   instHMISettings.instAniPNTmr.stations.me[24].kp8Config.colorOn1[0] := 'off';
   instHMISettings.instAniPNTmr.stations.me[24].kp8Config.colorOn1[1] := 'off';
   instHMISettings.instAniPNTmr.stations.me[24].kp8Config.colorOn1[2] := 'off';
   instHMISettings.instAniPNTmr.stations.me[24].kp8Config.colorOn1[3] := 'off';
   instHMISettings.instAniPNTmr.stations.me[24].kp8Config.colorOn1[4] := 'off';
   instHMISettings.instAniPNTmr.stations.me[24].kp8Config.colorOn1[5] := 'off';
   instHMISettings.instAniPNTmr.stations.me[24].kp8Config.colorOn1[6] := 'off';
   instHMISettings.instAniPNTmr.stations.me[24].kp8Config.colorOn1[7] := 'yellow';
   instHMISettings.instAniPNTmr.stations.me[24].kp8Config.colorOn2[0] := 'off';
   instHMISettings.instAniPNTmr.stations.me[24].kp8Config.colorOn2[1] := 'off';
   instHMISettings.instAniPNTmr.stations.me[24].kp8Config.colorOn2[2] := 'off';
   instHMISettings.instAniPNTmr.stations.me[24].kp8Config.colorOn2[3] := 'off';
   instHMISettings.instAniPNTmr.stations.me[24].kp8Config.colorOn2[4] := 'off';
   instHMISettings.instAniPNTmr.stations.me[24].kp8Config.colorOn2[5] := 'off';
   instHMISettings.instAniPNTmr.stations.me[24].kp8Config.colorOn2[6] := 'off';
   instHMISettings.instAniPNTmr.stations.me[24].kp8Config.colorOff[0] := 'off';
   instHMISettings.instAniPNTmr.stations.me[24].kp8Config.colorOff[1] := 'off';
   instHMISettings.instAniPNTmr.stations.me[24].kp8Config.colorOff[2] := 'off';
   instHMISettings.instAniPNTmr.stations.me[24].kp8Config.colorOff[3] := 'off';
   instHMISettings.instAniPNTmr.stations.me[24].kp8Config.colorOff[4] := 'off';
   instHMISettings.instAniPNTmr.stations.me[24].kp8Config.colorOff[5] := 'off';
   instHMISettings.instAniPNTmr.stations.me[24].kp8Config.colorOff[6] := 'off';
   instHMISettings.instAniPNTmr.stations.me[24].kp8Config.colorOff[7] := 'green';
   instHMISettings.instAniPNTmr.stations.me[24].kp8Config.mode[7] := TRUE;
   instHMISettings.instAniPNTmr.stations.me[24].kp8Out := 16#0080_0000;
   instHMISettings.instAniPNTmr.stations.me[24].line := WSTRING#'LGS';
   instHMISettings.instAniPNTmr.stations.me[24].partNumbers[0] := WSTRING#'';
   instHMISettings.instAniPNTmr.stations.me[24].partNumbers[1] := WSTRING#'';
   instHMISettings.instAniPNTmr.stations.me[24].partNumbers[2] := WSTRING#'';
   instHMISettings.instAniPNTmr.stations.me[24].partNumbers[3] := WSTRING#'';
   instHMISettings.instAniPNTmr.stations.me[24].partNumbers[4] := WSTRING#'';
   instHMISettings.instAniPNTmr.stations.me[24].partNumbers[5] := WSTRING#'';
   instHMISettings.instAniPNTmr.stations.me[24].partNumbers[6] := WSTRING#'';
   instHMISettings.instAniPNTmr.stations.me[24].partNumbers[7] := WSTRING#'16.08.208.411.030C';
   instHMISettings.instAniPNTmr.stations.me[24].presetTime.allotted[7] := 1800.0;
   instHMISettings.instAniPNTmr.stations.me[24].presetTime.critical[7] := 300.0;
   instHMISettings.instAniPNTmr.stations.me[24].stackLightOut := 16#0400_0000;
   instHMISettings.instAniPNTmr.stations.me[25].btnStates[0] := TRUE;
   instHMISettings.instAniPNTmr.stations.me[25].dropZone := 1;
   instHMISettings.instAniPNTmr.stations.me[25].kp8Config.activate[1] := TRUE;
   instHMISettings.instAniPNTmr.stations.me[25].kp8Config.activate[2] := TRUE;
   instHMISettings.instAniPNTmr.stations.me[25].kp8Config.activate[6] := TRUE;
   instHMISettings.instAniPNTmr.stations.me[25].kp8Config.activate[7] := TRUE;
   instHMISettings.instAniPNTmr.stations.me[25].kp8Config.colorOn1[0] := 'off';
   instHMISettings.instAniPNTmr.stations.me[25].kp8Config.colorOn1[1] := 'yellow';
   instHMISettings.instAniPNTmr.stations.me[25].kp8Config.colorOn1[2] := 'yellow';
   instHMISettings.instAniPNTmr.stations.me[25].kp8Config.colorOn1[3] := 'off';
   instHMISettings.instAniPNTmr.stations.me[25].kp8Config.colorOn1[4] := 'off';
   instHMISettings.instAniPNTmr.stations.me[25].kp8Config.colorOn1[5] := 'off';
   instHMISettings.instAniPNTmr.stations.me[25].kp8Config.colorOn1[6] := 'yellow';
   instHMISettings.instAniPNTmr.stations.me[25].kp8Config.colorOn1[7] := 'yellow';
   instHMISettings.instAniPNTmr.stations.me[25].kp8Config.colorOn2[0] := 'off';
   instHMISettings.instAniPNTmr.stations.me[25].kp8Config.colorOn2[3] := 'off';
   instHMISettings.instAniPNTmr.stations.me[25].kp8Config.colorOn2[4] := 'off';
   instHMISettings.instAniPNTmr.stations.me[25].kp8Config.colorOn2[5] := 'off';
   instHMISettings.instAniPNTmr.stations.me[25].kp8Config.colorOff[0] := 'off';
   instHMISettings.instAniPNTmr.stations.me[25].kp8Config.colorOff[1] := 'green';
   instHMISettings.instAniPNTmr.stations.me[25].kp8Config.colorOff[2] := 'green';
   instHMISettings.instAniPNTmr.stations.me[25].kp8Config.colorOff[3] := 'off';
   instHMISettings.instAniPNTmr.stations.me[25].kp8Config.colorOff[4] := 'off';
   instHMISettings.instAniPNTmr.stations.me[25].kp8Config.colorOff[5] := 'off';
   instHMISettings.instAniPNTmr.stations.me[25].kp8Config.colorOff[6] := 'green';
   instHMISettings.instAniPNTmr.stations.me[25].kp8Config.colorOff[7] := 'green';
   instHMISettings.instAniPNTmr.stations.me[25].kp8Config.mode[1] := TRUE;
   instHMISettings.instAniPNTmr.stations.me[25].kp8Config.mode[2] := TRUE;
   instHMISettings.instAniPNTmr.stations.me[25].kp8Config.mode[6] := TRUE;
   instHMISettings.instAniPNTmr.stations.me[25].kp8Config.mode[7] := TRUE;
   instHMISettings.instAniPNTmr.stations.me[25].kp8Out := 16#4000_8400;
   instHMISettings.instAniPNTmr.stations.me[25].line := WSTRING#'CV';
   instHMISettings.instAniPNTmr.stations.me[25].partNumbers[0] := WSTRING#'';
   instHMISettings.instAniPNTmr.stations.me[25].partNumbers[1] := WSTRING#'C/O MATERIALS';
   instHMISettings.instAniPNTmr.stations.me[25].partNumbers[2] := WSTRING#'16.08.216.806.020A';
   instHMISettings.instAniPNTmr.stations.me[25].partNumbers[3] := WSTRING#'';
   instHMISettings.instAniPNTmr.stations.me[25].partNumbers[4] := WSTRING#'';
   instHMISettings.instAniPNTmr.stations.me[25].partNumbers[5] := WSTRING#'';
   instHMISettings.instAniPNTmr.stations.me[25].partNumbers[6] := WSTRING#'16.08.208.631.000F';
   instHMISettings.instAniPNTmr.stations.me[25].partNumbers[7] := WSTRING#'16.08.216.315.000A';
   instHMISettings.instAniPNTmr.stations.me[25].presetTime.allotted[1] := 1800.0;
   instHMISettings.instAniPNTmr.stations.me[25].presetTime.allotted[2] := 1800.0;
   instHMISettings.instAniPNTmr.stations.me[25].presetTime.allotted[6] := 1800.0;
   instHMISettings.instAniPNTmr.stations.me[25].presetTime.allotted[7] := 1800.0;
   instHMISettings.instAniPNTmr.stations.me[25].presetTime.critical[1] := 300.0;
   instHMISettings.instAniPNTmr.stations.me[25].presetTime.critical[2] := 300.0;
   instHMISettings.instAniPNTmr.stations.me[25].presetTime.critical[6] := 300.0;
   instHMISettings.instAniPNTmr.stations.me[25].presetTime.critical[7] := 300.0;
   instHMISettings.instAniPNTmr.stations.me[25].settings.btnSelection[1] := TRUE;
   instHMISettings.instAniPNTmr.stations.me[25].stackLightOut := 16#0409_0200;
   instHMISettings.instAniPNTmr.stations.me[26].animations[3] := 3;
   instHMISettings.instAniPNTmr.stations.me[26].btnStates[3] := TRUE;
   instHMISettings.instAniPNTmr.stations.me[26].dropZone := 2;
   instHMISettings.instAniPNTmr.stations.me[26].elapsedTime.partReq[3] := 2305.587;
   instHMISettings.instAniPNTmr.stations.me[26].kp8Config.activate[1] := TRUE;
   instHMISettings.instAniPNTmr.stations.me[26].kp8Config.activate[2] := TRUE;
   instHMISettings.instAniPNTmr.stations.me[26].kp8Config.activate[3] := TRUE;
   instHMISettings.instAniPNTmr.stations.me[26].kp8Config.activate[5] := TRUE;
   instHMISettings.instAniPNTmr.stations.me[26].kp8Config.activate[6] := TRUE;
   instHMISettings.instAniPNTmr.stations.me[26].kp8Config.activate[7] := TRUE;
   instHMISettings.instAniPNTmr.stations.me[26].kp8Config.colorOn1[0] := 'off';
   instHMISettings.instAniPNTmr.stations.me[26].kp8Config.colorOn1[1] := 'yellow';
   instHMISettings.instAniPNTmr.stations.me[26].kp8Config.colorOn1[2] := 'yellow';
   instHMISettings.instAniPNTmr.stations.me[26].kp8Config.colorOn1[3] := 'yellow';
   instHMISettings.instAniPNTmr.stations.me[26].kp8Config.colorOn1[4] := 'off';
   instHMISettings.instAniPNTmr.stations.me[26].kp8Config.colorOn1[5] := 'yellow';
   instHMISettings.instAniPNTmr.stations.me[26].kp8Config.colorOn1[6] := 'yellow';
   instHMISettings.instAniPNTmr.stations.me[26].kp8Config.colorOn1[7] := 'yellow';
   instHMISettings.instAniPNTmr.stations.me[26].kp8Config.colorOn2[0] := 'off';
   instHMISettings.instAniPNTmr.stations.me[26].kp8Config.colorOn2[4] := 'off';
   instHMISettings.instAniPNTmr.stations.me[26].kp8Config.colorOff[0] := 'off';
   instHMISettings.instAniPNTmr.stations.me[26].kp8Config.colorOff[1] := 'green';
   instHMISettings.instAniPNTmr.stations.me[26].kp8Config.colorOff[2] := 'green';
   instHMISettings.instAniPNTmr.stations.me[26].kp8Config.colorOff[3] := 'green';
   instHMISettings.instAniPNTmr.stations.me[26].kp8Config.colorOff[4] := 'off';
   instHMISettings.instAniPNTmr.stations.me[26].kp8Config.colorOff[5] := 'green';
   instHMISettings.instAniPNTmr.stations.me[26].kp8Config.colorOff[6] := 'green';
   instHMISettings.instAniPNTmr.stations.me[26].kp8Config.colorOff[7] := 'green';
   instHMISettings.instAniPNTmr.stations.me[26].kp8Config.mode[1] := TRUE;
   instHMISettings.instAniPNTmr.stations.me[26].kp8Config.mode[2] := TRUE;
   instHMISettings.instAniPNTmr.stations.me[26].kp8Config.mode[3] := TRUE;
   instHMISettings.instAniPNTmr.stations.me[26].kp8Config.mode[5] := TRUE;
   instHMISettings.instAniPNTmr.stations.me[26].kp8Config.mode[6] := TRUE;
   instHMISettings.instAniPNTmr.stations.me[26].kp8Config.mode[7] := TRUE;
   instHMISettings.instAniPNTmr.stations.me[26].kp8Out := 16#E000_0000;
   instHMISettings.instAniPNTmr.stations.me[26].line := WSTRING#'CV';
   instHMISettings.instAniPNTmr.stations.me[26].partNumbers[0] := WSTRING#'';
   instHMISettings.instAniPNTmr.stations.me[26].partNumbers[1] := WSTRING#'C/O MATERIALS';
   instHMISettings.instAniPNTmr.stations.me[26].partNumbers[2] := WSTRING#'16.08.216.291.000A';
   instHMISettings.instAniPNTmr.stations.me[26].partNumbers[3] := WSTRING#'16.08.216.315.001A';
   instHMISettings.instAniPNTmr.stations.me[26].partNumbers[4] := WSTRING#'';
   instHMISettings.instAniPNTmr.stations.me[26].partNumbers[5] := WSTRING#'16.08.216.057.001A';
   instHMISettings.instAniPNTmr.stations.me[26].partNumbers[6] := WSTRING#'16.08.208.661.000F';
   instHMISettings.instAniPNTmr.stations.me[26].partNumbers[7] := WSTRING#'16.08.216.315.002A';
   instHMISettings.instAniPNTmr.stations.me[26].partOrdered[3] := TRUE;
   instHMISettings.instAniPNTmr.stations.me[26].partRequested[3] := TRUE;
   instHMISettings.instAniPNTmr.stations.me[26].presetTime.allotted[1] := 1800.0;
   instHMISettings.instAniPNTmr.stations.me[26].presetTime.allotted[2] := 1800.0;
   instHMISettings.instAniPNTmr.stations.me[26].presetTime.allotted[3] := 1800.0;
   instHMISettings.instAniPNTmr.stations.me[26].presetTime.allotted[5] := 1800.0;
   instHMISettings.instAniPNTmr.stations.me[26].presetTime.allotted[6] := 1800.0;
   instHMISettings.instAniPNTmr.stations.me[26].presetTime.allotted[7] := 1800.0;
   instHMISettings.instAniPNTmr.stations.me[26].presetTime.critical[1] := 300.0;
   instHMISettings.instAniPNTmr.stations.me[26].presetTime.critical[2] := 300.0;
   instHMISettings.instAniPNTmr.stations.me[26].presetTime.critical[3] := 300.0;
   instHMISettings.instAniPNTmr.stations.me[26].presetTime.critical[5] := 300.0;
   instHMISettings.instAniPNTmr.stations.me[26].presetTime.critical[6] := 300.0;
   instHMISettings.instAniPNTmr.stations.me[26].presetTime.critical[7] := 300.0;
   instHMISettings.instAniPNTmr.stations.me[26].stackLightOut := 16#0449_0200;
   instHMISettings.instAniPNTmr.stations.me[27].dropZone := 3;
   instHMISettings.instAniPNTmr.stations.me[27].kp8Config.activate[1] := TRUE;
   instHMISettings.instAniPNTmr.stations.me[27].kp8Config.activate[2] := TRUE;
   instHMISettings.instAniPNTmr.stations.me[27].kp8Config.activate[3] := TRUE;
   instHMISettings.instAniPNTmr.stations.me[27].kp8Config.activate[5] := TRUE;
   instHMISettings.instAniPNTmr.stations.me[27].kp8Config.activate[6] := TRUE;
   instHMISettings.instAniPNTmr.stations.me[27].kp8Config.activate[7] := TRUE;
   instHMISettings.instAniPNTmr.stations.me[27].kp8Config.colorOn1[0] := 'off';
   instHMISettings.instAniPNTmr.stations.me[27].kp8Config.colorOn1[1] := 'yellow';
   instHMISettings.instAniPNTmr.stations.me[27].kp8Config.colorOn1[2] := 'yellow';
   instHMISettings.instAniPNTmr.stations.me[27].kp8Config.colorOn1[3] := 'yellow';
   instHMISettings.instAniPNTmr.stations.me[27].kp8Config.colorOn1[4] := 'off';
   instHMISettings.instAniPNTmr.stations.me[27].kp8Config.colorOn1[5] := 'yellow';
   instHMISettings.instAniPNTmr.stations.me[27].kp8Config.colorOn1[6] := 'yellow';
   instHMISettings.instAniPNTmr.stations.me[27].kp8Config.colorOn1[7] := 'yellow';
   instHMISettings.instAniPNTmr.stations.me[27].kp8Config.colorOn2[0] := 'off';
   instHMISettings.instAniPNTmr.stations.me[27].kp8Config.colorOn2[4] := 'off';
   instHMISettings.instAniPNTmr.stations.me[27].kp8Config.colorOff[0] := 'off';
   instHMISettings.instAniPNTmr.stations.me[27].kp8Config.colorOff[1] := 'green';
   instHMISettings.instAniPNTmr.stations.me[27].kp8Config.colorOff[2] := 'green';
   instHMISettings.instAniPNTmr.stations.me[27].kp8Config.colorOff[3] := 'green';
   instHMISettings.instAniPNTmr.stations.me[27].kp8Config.colorOff[4] := 'off';
   instHMISettings.instAniPNTmr.stations.me[27].kp8Config.colorOff[5] := 'green';
   instHMISettings.instAniPNTmr.stations.me[27].kp8Config.colorOff[6] := 'green';
   instHMISettings.instAniPNTmr.stations.me[27].kp8Config.colorOff[7] := 'green';
   instHMISettings.instAniPNTmr.stations.me[27].kp8Config.mode[1] := TRUE;
   instHMISettings.instAniPNTmr.stations.me[27].kp8Config.mode[2] := TRUE;
   instHMISettings.instAniPNTmr.stations.me[27].kp8Config.mode[3] := TRUE;
   instHMISettings.instAniPNTmr.stations.me[27].kp8Config.mode[5] := TRUE;
   instHMISettings.instAniPNTmr.stations.me[27].kp8Config.mode[6] := TRUE;
   instHMISettings.instAniPNTmr.stations.me[27].kp8Config.mode[7] := TRUE;
   instHMISettings.instAniPNTmr.stations.me[27].kp8Out := 16#4000_A800;
   instHMISettings.instAniPNTmr.stations.me[27].line := WSTRING#'CV';
   instHMISettings.instAniPNTmr.stations.me[27].partNumbers[0] := WSTRING#'';
   instHMISettings.instAniPNTmr.stations.me[27].partNumbers[1] := WSTRING#'C/O MATERIALS';
   instHMISettings.instAniPNTmr.stations.me[27].partNumbers[2] := WSTRING#'16.18.011.301.010A';
   instHMISettings.instAniPNTmr.stations.me[27].partNumbers[3] := WSTRING#'16.18.011.301.020B';
   instHMISettings.instAniPNTmr.stations.me[27].partNumbers[4] := WSTRING#'';
   instHMISettings.instAniPNTmr.stations.me[27].partNumbers[5] := WSTRING#'16.18.007.311.010A';
   instHMISettings.instAniPNTmr.stations.me[27].partNumbers[6] := WSTRING#'16.18.007.311.020A';
   instHMISettings.instAniPNTmr.stations.me[27].partNumbers[7] := WSTRING#'16.18.012.401.020A';
   instHMISettings.instAniPNTmr.stations.me[27].presetTime.allotted[1] := 1800.0;
   instHMISettings.instAniPNTmr.stations.me[27].presetTime.allotted[2] := 1800.0;
   instHMISettings.instAniPNTmr.stations.me[27].presetTime.allotted[3] := 1800.0;
   instHMISettings.instAniPNTmr.stations.me[27].presetTime.allotted[5] := 1800.0;
   instHMISettings.instAniPNTmr.stations.me[27].presetTime.allotted[6] := 1800.0;
   instHMISettings.instAniPNTmr.stations.me[27].presetTime.allotted[7] := 1800.0;
   instHMISettings.instAniPNTmr.stations.me[27].presetTime.critical[1] := 300.0;
   instHMISettings.instAniPNTmr.stations.me[27].presetTime.critical[2] := 300.0;
   instHMISettings.instAniPNTmr.stations.me[27].presetTime.critical[3] := 300.0;
   instHMISettings.instAniPNTmr.stations.me[27].presetTime.critical[5] := 300.0;
   instHMISettings.instAniPNTmr.stations.me[27].presetTime.critical[6] := 300.0;
   instHMISettings.instAniPNTmr.stations.me[27].presetTime.critical[7] := 300.0;
   instHMISettings.instAniPNTmr.stations.me[27].stackLightOut := 16#2449_0200;
   instHMISettings.instAniPNTmr.stations.me[28].dropZone := 4;
   instHMISettings.instAniPNTmr.stations.me[28].kp8Config.activate[1] := TRUE;
   instHMISettings.instAniPNTmr.stations.me[28].kp8Config.activate[3] := TRUE;
   instHMISettings.instAniPNTmr.stations.me[28].kp8Config.activate[6] := TRUE;
   instHMISettings.instAniPNTmr.stations.me[28].kp8Config.activate[7] := TRUE;
   instHMISettings.instAniPNTmr.stations.me[28].kp8Config.colorOn1[0] := 'off';
   instHMISettings.instAniPNTmr.stations.me[28].kp8Config.colorOn1[1] := 'yellow';
   instHMISettings.instAniPNTmr.stations.me[28].kp8Config.colorOn1[2] := 'off';
   instHMISettings.instAniPNTmr.stations.me[28].kp8Config.colorOn1[3] := 'yellow';
   instHMISettings.instAniPNTmr.stations.me[28].kp8Config.colorOn1[4] := 'off';
   instHMISettings.instAniPNTmr.stations.me[28].kp8Config.colorOn1[5] := 'off';
   instHMISettings.instAniPNTmr.stations.me[28].kp8Config.colorOn1[6] := 'yellow';
   instHMISettings.instAniPNTmr.stations.me[28].kp8Config.colorOn1[7] := 'yellow';
   instHMISettings.instAniPNTmr.stations.me[28].kp8Config.colorOn2[0] := 'off';
   instHMISettings.instAniPNTmr.stations.me[28].kp8Config.colorOn2[2] := 'off';
   instHMISettings.instAniPNTmr.stations.me[28].kp8Config.colorOn2[4] := 'off';
   instHMISettings.instAniPNTmr.stations.me[28].kp8Config.colorOn2[5] := 'off';
   instHMISettings.instAniPNTmr.stations.me[28].kp8Config.colorOff[0] := 'off';
   instHMISettings.instAniPNTmr.stations.me[28].kp8Config.colorOff[1] := 'green';
   instHMISettings.instAniPNTmr.stations.me[28].kp8Config.colorOff[2] := 'off';
   instHMISettings.instAniPNTmr.stations.me[28].kp8Config.colorOff[3] := 'green';
   instHMISettings.instAniPNTmr.stations.me[28].kp8Config.colorOff[4] := 'off';
   instHMISettings.instAniPNTmr.stations.me[28].kp8Config.colorOff[5] := 'off';
   instHMISettings.instAniPNTmr.stations.me[28].kp8Config.colorOff[6] := 'green';
   instHMISettings.instAniPNTmr.stations.me[28].kp8Config.colorOff[7] := 'green';
   instHMISettings.instAniPNTmr.stations.me[28].kp8Config.mode[1] := TRUE;
   instHMISettings.instAniPNTmr.stations.me[28].kp8Config.mode[3] := TRUE;
   instHMISettings.instAniPNTmr.stations.me[28].kp8Config.mode[6] := TRUE;
   instHMISettings.instAniPNTmr.stations.me[28].kp8Config.mode[7] := TRUE;
   instHMISettings.instAniPNTmr.stations.me[28].kp8Out := 16#0000_6E00;
   instHMISettings.instAniPNTmr.stations.me[28].line := WSTRING#'CV';
   instHMISettings.instAniPNTmr.stations.me[28].partNumbers[0] := WSTRING#'';
   instHMISettings.instAniPNTmr.stations.me[28].partNumbers[1] := WSTRING#'C/O MATERIALS';
   instHMISettings.instAniPNTmr.stations.me[28].partNumbers[2] := WSTRING#'';
   instHMISettings.instAniPNTmr.stations.me[28].partNumbers[3] := WSTRING#'16.32.112.543.210E';
   instHMISettings.instAniPNTmr.stations.me[28].partNumbers[4] := WSTRING#'';
   instHMISettings.instAniPNTmr.stations.me[28].partNumbers[5] := WSTRING#'';
   instHMISettings.instAniPNTmr.stations.me[28].partNumbers[6] := WSTRING#'16.32.112.543.020A';
   instHMISettings.instAniPNTmr.stations.me[28].partNumbers[7] := WSTRING#'16.32.112.315.018A';
   instHMISettings.instAniPNTmr.stations.me[28].presetTime.allotted[1] := 1800.0;
   instHMISettings.instAniPNTmr.stations.me[28].presetTime.allotted[3] := 1800.0;
   instHMISettings.instAniPNTmr.stations.me[28].presetTime.allotted[6] := 1800.0;
   instHMISettings.instAniPNTmr.stations.me[28].presetTime.allotted[7] := 1800.0;
   instHMISettings.instAniPNTmr.stations.me[28].presetTime.critical[1] := 300.0;
   instHMISettings.instAniPNTmr.stations.me[28].presetTime.critical[3] := 300.0;
   instHMISettings.instAniPNTmr.stations.me[28].presetTime.critical[6] := 300.0;
   instHMISettings.instAniPNTmr.stations.me[28].presetTime.critical[7] := 300.0;
   instHMISettings.instAniPNTmr.stations.me[28].stackLightOut := 16#2401_0200;
   instHMISettings.instAniPNTmr.stations.me[29].dropZone := 1;
   instHMISettings.instAniPNTmr.stations.me[29].kp8Config.activate[1] := TRUE;
   instHMISettings.instAniPNTmr.stations.me[29].kp8Config.activate[2] := TRUE;
   instHMISettings.instAniPNTmr.stations.me[29].kp8Config.activate[3] := TRUE;
   instHMISettings.instAniPNTmr.stations.me[29].kp8Config.activate[5] := TRUE;
   instHMISettings.instAniPNTmr.stations.me[29].kp8Config.activate[6] := TRUE;
   instHMISettings.instAniPNTmr.stations.me[29].kp8Config.activate[7] := TRUE;
   instHMISettings.instAniPNTmr.stations.me[29].kp8Config.colorOn1[0] := 'off';
   instHMISettings.instAniPNTmr.stations.me[29].kp8Config.colorOn1[1] := 'yellow';
   instHMISettings.instAniPNTmr.stations.me[29].kp8Config.colorOn1[2] := 'yellow';
   instHMISettings.instAniPNTmr.stations.me[29].kp8Config.colorOn1[3] := 'yellow';
   instHMISettings.instAniPNTmr.stations.me[29].kp8Config.colorOn1[4] := 'off';
   instHMISettings.instAniPNTmr.stations.me[29].kp8Config.colorOn1[5] := 'yellow';
   instHMISettings.instAniPNTmr.stations.me[29].kp8Config.colorOn1[6] := 'yellow';
   instHMISettings.instAniPNTmr.stations.me[29].kp8Config.colorOn1[7] := 'yellow';
   instHMISettings.instAniPNTmr.stations.me[29].kp8Config.colorOn2[0] := 'off';
   instHMISettings.instAniPNTmr.stations.me[29].kp8Config.colorOn2[4] := 'off';
   instHMISettings.instAniPNTmr.stations.me[29].kp8Config.colorOff[0] := 'off';
   instHMISettings.instAniPNTmr.stations.me[29].kp8Config.colorOff[1] := 'green';
   instHMISettings.instAniPNTmr.stations.me[29].kp8Config.colorOff[2] := 'green';
   instHMISettings.instAniPNTmr.stations.me[29].kp8Config.colorOff[3] := 'green';
   instHMISettings.instAniPNTmr.stations.me[29].kp8Config.colorOff[4] := 'off';
   instHMISettings.instAniPNTmr.stations.me[29].kp8Config.colorOff[5] := 'green';
   instHMISettings.instAniPNTmr.stations.me[29].kp8Config.colorOff[6] := 'green';
   instHMISettings.instAniPNTmr.stations.me[29].kp8Config.colorOff[7] := 'green';
   instHMISettings.instAniPNTmr.stations.me[29].kp8Config.mode[1] := TRUE;
   instHMISettings.instAniPNTmr.stations.me[29].kp8Config.mode[2] := TRUE;
   instHMISettings.instAniPNTmr.stations.me[29].kp8Config.mode[3] := TRUE;
   instHMISettings.instAniPNTmr.stations.me[29].kp8Config.mode[5] := TRUE;
   instHMISettings.instAniPNTmr.stations.me[29].kp8Config.mode[6] := TRUE;
   instHMISettings.instAniPNTmr.stations.me[29].kp8Config.mode[7] := TRUE;
   instHMISettings.instAniPNTmr.stations.me[29].kp8Out := 16#2A00_4400;
   instHMISettings.instAniPNTmr.stations.me[29].line := WSTRING#'PC';
   instHMISettings.instAniPNTmr.stations.me[29].partNumbers[0] := WSTRING#'';
   instHMISettings.instAniPNTmr.stations.me[29].partNumbers[1] := WSTRING#'C/O MATERIALS';
   instHMISettings.instAniPNTmr.stations.me[29].partNumbers[2] := WSTRING#'11.54.007.052.007B';
   instHMISettings.instAniPNTmr.stations.me[29].partNumbers[3] := WSTRING#'11.54.007.315.026G';
   instHMISettings.instAniPNTmr.stations.me[29].partNumbers[4] := WSTRING#'';
   instHMISettings.instAniPNTmr.stations.me[29].partNumbers[5] := WSTRING#'11.54.007.052.008A';
   instHMISettings.instAniPNTmr.stations.me[29].partNumbers[6] := WSTRING#'11.54.007.045.015D';
   instHMISettings.instAniPNTmr.stations.me[29].partNumbers[7] := WSTRING#'11.54.017.315.001F';
   instHMISettings.instAniPNTmr.stations.me[29].presetTime.allotted[1] := 1800.0;
   instHMISettings.instAniPNTmr.stations.me[29].presetTime.allotted[2] := 1800.0;
   instHMISettings.instAniPNTmr.stations.me[29].presetTime.allotted[3] := 1800.0;
   instHMISettings.instAniPNTmr.stations.me[29].presetTime.allotted[5] := 1800.0;
   instHMISettings.instAniPNTmr.stations.me[29].presetTime.allotted[6] := 1800.0;
   instHMISettings.instAniPNTmr.stations.me[29].presetTime.allotted[7] := 1800.0;
   instHMISettings.instAniPNTmr.stations.me[29].presetTime.critical[1] := 300.0;
   instHMISettings.instAniPNTmr.stations.me[29].presetTime.critical[2] := 300.0;
   instHMISettings.instAniPNTmr.stations.me[29].presetTime.critical[3] := 300.0;
   instHMISettings.instAniPNTmr.stations.me[29].presetTime.critical[5] := 300.0;
   instHMISettings.instAniPNTmr.stations.me[29].presetTime.critical[6] := 300.0;
   instHMISettings.instAniPNTmr.stations.me[29].presetTime.critical[7] := 300.0;
   instHMISettings.instAniPNTmr.stations.me[29].settings.btnSelection[3] := TRUE;
   instHMISettings.instAniPNTmr.stations.me[29].stackLightOut := 16#2449_0200;
   instHMISettings.instAniPNTmr.stations.me[30].dropZone := 1;
   instHMISettings.instAniPNTmr.stations.me[30].kp8Config.activate[7] := TRUE;
   instHMISettings.instAniPNTmr.stations.me[30].kp8Config.colorOn1[0] := 'off';
   instHMISettings.instAniPNTmr.stations.me[30].kp8Config.colorOn1[1] := 'off';
   instHMISettings.instAniPNTmr.stations.me[30].kp8Config.colorOn1[2] := 'off';
   instHMISettings.instAniPNTmr.stations.me[30].kp8Config.colorOn1[3] := 'off';
   instHMISettings.instAniPNTmr.stations.me[30].kp8Config.colorOn1[4] := 'off';
   instHMISettings.instAniPNTmr.stations.me[30].kp8Config.colorOn1[5] := 'off';
   instHMISettings.instAniPNTmr.stations.me[30].kp8Config.colorOn1[6] := 'off';
   instHMISettings.instAniPNTmr.stations.me[30].kp8Config.colorOn1[7] := 'yellow';
   instHMISettings.instAniPNTmr.stations.me[30].kp8Config.colorOn2[0] := 'off';
   instHMISettings.instAniPNTmr.stations.me[30].kp8Config.colorOn2[1] := 'off';
   instHMISettings.instAniPNTmr.stations.me[30].kp8Config.colorOn2[2] := 'off';
   instHMISettings.instAniPNTmr.stations.me[30].kp8Config.colorOn2[3] := 'off';
   instHMISettings.instAniPNTmr.stations.me[30].kp8Config.colorOn2[4] := 'off';
   instHMISettings.instAniPNTmr.stations.me[30].kp8Config.colorOn2[5] := 'off';
   instHMISettings.instAniPNTmr.stations.me[30].kp8Config.colorOn2[6] := 'off';
   instHMISettings.instAniPNTmr.stations.me[30].kp8Config.colorOff[0] := 'off';
   instHMISettings.instAniPNTmr.stations.me[30].kp8Config.colorOff[1] := 'off';
   instHMISettings.instAniPNTmr.stations.me[30].kp8Config.colorOff[2] := 'off';
   instHMISettings.instAniPNTmr.stations.me[30].kp8Config.colorOff[3] := 'off';
   instHMISettings.instAniPNTmr.stations.me[30].kp8Config.colorOff[4] := 'off';
   instHMISettings.instAniPNTmr.stations.me[30].kp8Config.colorOff[5] := 'off';
   instHMISettings.instAniPNTmr.stations.me[30].kp8Config.colorOff[6] := 'off';
   instHMISettings.instAniPNTmr.stations.me[30].kp8Config.colorOff[7] := 'green';
   instHMISettings.instAniPNTmr.stations.me[30].kp8Config.mode[7] := TRUE;
   instHMISettings.instAniPNTmr.stations.me[30].kp8Out := 16#0080_0000;
   instHMISettings.instAniPNTmr.stations.me[30].line := WSTRING#'VN127';
   instHMISettings.instAniPNTmr.stations.me[30].partNumbers[0] := WSTRING#'';
   instHMISettings.instAniPNTmr.stations.me[30].partNumbers[1] := WSTRING#'';
   instHMISettings.instAniPNTmr.stations.me[30].partNumbers[2] := WSTRING#'';
   instHMISettings.instAniPNTmr.stations.me[30].partNumbers[3] := WSTRING#'';
   instHMISettings.instAniPNTmr.stations.me[30].partNumbers[4] := WSTRING#'';
   instHMISettings.instAniPNTmr.stations.me[30].partNumbers[5] := WSTRING#'';
   instHMISettings.instAniPNTmr.stations.me[30].partNumbers[6] := WSTRING#'';
   instHMISettings.instAniPNTmr.stations.me[30].partNumbers[7] := WSTRING#'11.54.313.872.000E';
   instHMISettings.instAniPNTmr.stations.me[30].presetTime.allotted[7] := 1800.0;
   instHMISettings.instAniPNTmr.stations.me[30].presetTime.critical[7] := 300.0;
   instHMISettings.instAniPNTmr.stations.me[30].settings.btnSelection[7] := TRUE;
   instHMISettings.instAniPNTmr.stations.me[30].stackLightOut := 16#0400_0000;
   instHMISettings.instAniPNTmr.stations.me[31].dropZone := 1;
   instHMISettings.instAniPNTmr.stations.me[31].kp8Config.activate[3] := TRUE;
   instHMISettings.instAniPNTmr.stations.me[31].kp8Config.activate[7] := TRUE;
   instHMISettings.instAniPNTmr.stations.me[31].kp8Config.colorOn1[0] := 'off';
   instHMISettings.instAniPNTmr.stations.me[31].kp8Config.colorOn1[1] := 'off';
   instHMISettings.instAniPNTmr.stations.me[31].kp8Config.colorOn1[2] := 'off';
   instHMISettings.instAniPNTmr.stations.me[31].kp8Config.colorOn1[3] := 'yellow';
   instHMISettings.instAniPNTmr.stations.me[31].kp8Config.colorOn1[4] := 'off';
   instHMISettings.instAniPNTmr.stations.me[31].kp8Config.colorOn1[5] := 'off';
   instHMISettings.instAniPNTmr.stations.me[31].kp8Config.colorOn1[6] := 'off';
   instHMISettings.instAniPNTmr.stations.me[31].kp8Config.colorOn1[7] := 'yellow';
   instHMISettings.instAniPNTmr.stations.me[31].kp8Config.colorOn2[0] := 'off';
   instHMISettings.instAniPNTmr.stations.me[31].kp8Config.colorOn2[1] := 'off';
   instHMISettings.instAniPNTmr.stations.me[31].kp8Config.colorOn2[2] := 'off';
   instHMISettings.instAniPNTmr.stations.me[31].kp8Config.colorOn2[4] := 'off';
   instHMISettings.instAniPNTmr.stations.me[31].kp8Config.colorOn2[5] := 'off';
   instHMISettings.instAniPNTmr.stations.me[31].kp8Config.colorOn2[6] := 'off';
   instHMISettings.instAniPNTmr.stations.me[31].kp8Config.colorOff[0] := 'off';
   instHMISettings.instAniPNTmr.stations.me[31].kp8Config.colorOff[1] := 'off';
   instHMISettings.instAniPNTmr.stations.me[31].kp8Config.colorOff[2] := 'off';
   instHMISettings.instAniPNTmr.stations.me[31].kp8Config.colorOff[3] := 'green';
   instHMISettings.instAniPNTmr.stations.me[31].kp8Config.colorOff[4] := 'off';
   instHMISettings.instAniPNTmr.stations.me[31].kp8Config.colorOff[5] := 'off';
   instHMISettings.instAniPNTmr.stations.me[31].kp8Config.colorOff[6] := 'off';
   instHMISettings.instAniPNTmr.stations.me[31].kp8Config.colorOff[7] := 'green';
   instHMISettings.instAniPNTmr.stations.me[31].kp8Config.mode[3] := TRUE;
   instHMISettings.instAniPNTmr.stations.me[31].kp8Config.mode[7] := TRUE;
   instHMISettings.instAniPNTmr.stations.me[31].kp8Out := 16#0088_0000;
   instHMISettings.instAniPNTmr.stations.me[31].line := WSTRING#'1BX 2.0';
   instHMISettings.instAniPNTmr.stations.me[31].partNumbers[0] := WSTRING#'';
   instHMISettings.instAniPNTmr.stations.me[31].partNumbers[1] := WSTRING#'';
   instHMISettings.instAniPNTmr.stations.me[31].partNumbers[2] := WSTRING#'';
   instHMISettings.instAniPNTmr.stations.me[31].partNumbers[3] := WSTRING#'16.08.216.011.030B';
   instHMISettings.instAniPNTmr.stations.me[31].partNumbers[4] := WSTRING#'';
   instHMISettings.instAniPNTmr.stations.me[31].partNumbers[5] := WSTRING#'';
   instHMISettings.instAniPNTmr.stations.me[31].partNumbers[6] := WSTRING#'';
   instHMISettings.instAniPNTmr.stations.me[31].partNumbers[7] := WSTRING#'16.08.208.161.030E';
   instHMISettings.instAniPNTmr.stations.me[31].presetTime.allotted[3] := 1800.0;
   instHMISettings.instAniPNTmr.stations.me[31].presetTime.allotted[7] := 1800.0;
   instHMISettings.instAniPNTmr.stations.me[31].presetTime.critical[3] := 300.0;
   instHMISettings.instAniPNTmr.stations.me[31].presetTime.critical[7] := 300.0;
   instHMISettings.instAniPNTmr.stations.me[31].stackLightOut := 16#2400_0000;
   instHMISettings.instAniPNTmr.stations.me[32].dropZone := 2;
   instHMISettings.instAniPNTmr.stations.me[32].kp8Config.activate[7] := TRUE;
   instHMISettings.instAniPNTmr.stations.me[32].kp8Config.colorOn1[0] := 'off';
   instHMISettings.instAniPNTmr.stations.me[32].kp8Config.colorOn1[1] := 'off';
   instHMISettings.instAniPNTmr.stations.me[32].kp8Config.colorOn1[2] := 'off';
   instHMISettings.instAniPNTmr.stations.me[32].kp8Config.colorOn1[3] := 'off';
   instHMISettings.instAniPNTmr.stations.me[32].kp8Config.colorOn1[4] := 'off';
   instHMISettings.instAniPNTmr.stations.me[32].kp8Config.colorOn1[5] := 'off';
   instHMISettings.instAniPNTmr.stations.me[32].kp8Config.colorOn1[6] := 'off';
   instHMISettings.instAniPNTmr.stations.me[32].kp8Config.colorOn1[7] := 'yellow';
   instHMISettings.instAniPNTmr.stations.me[32].kp8Config.colorOn2[0] := 'off';
   instHMISettings.instAniPNTmr.stations.me[32].kp8Config.colorOn2[1] := 'off';
   instHMISettings.instAniPNTmr.stations.me[32].kp8Config.colorOn2[2] := 'off';
   instHMISettings.instAniPNTmr.stations.me[32].kp8Config.colorOn2[3] := 'off';
   instHMISettings.instAniPNTmr.stations.me[32].kp8Config.colorOn2[4] := 'off';
   instHMISettings.instAniPNTmr.stations.me[32].kp8Config.colorOn2[5] := 'off';
   instHMISettings.instAniPNTmr.stations.me[32].kp8Config.colorOn2[6] := 'off';
   instHMISettings.instAniPNTmr.stations.me[32].kp8Config.colorOff[0] := 'off';
   instHMISettings.instAniPNTmr.stations.me[32].kp8Config.colorOff[1] := 'off';
   instHMISettings.instAniPNTmr.stations.me[32].kp8Config.colorOff[2] := 'off';
   instHMISettings.instAniPNTmr.stations.me[32].kp8Config.colorOff[3] := 'off';
   instHMISettings.instAniPNTmr.stations.me[32].kp8Config.colorOff[4] := 'off';
   instHMISettings.instAniPNTmr.stations.me[32].kp8Config.colorOff[5] := 'off';
   instHMISettings.instAniPNTmr.stations.me[32].kp8Config.colorOff[6] := 'off';
   instHMISettings.instAniPNTmr.stations.me[32].kp8Config.colorOff[7] := 'green';
   instHMISettings.instAniPNTmr.stations.me[32].kp8Config.mode[7] := TRUE;
   instHMISettings.instAniPNTmr.stations.me[32].kp8Out := 16#0080_0000;
   instHMISettings.instAniPNTmr.stations.me[32].line := WSTRING#'1BX 2.0';
   instHMISettings.instAniPNTmr.stations.me[32].partNumbers[0] := WSTRING#'';
   instHMISettings.instAniPNTmr.stations.me[32].partNumbers[1] := WSTRING#'';
   instHMISettings.instAniPNTmr.stations.me[32].partNumbers[2] := WSTRING#'';
   instHMISettings.instAniPNTmr.stations.me[32].partNumbers[3] := WSTRING#'';
   instHMISettings.instAniPNTmr.stations.me[32].partNumbers[4] := WSTRING#'';
   instHMISettings.instAniPNTmr.stations.me[32].partNumbers[5] := WSTRING#'';
   instHMISettings.instAniPNTmr.stations.me[32].partNumbers[6] := WSTRING#'';
   instHMISettings.instAniPNTmr.stations.me[32].partNumbers[7] := WSTRING#'16.08.208.601.010D';
   instHMISettings.instAniPNTmr.stations.me[32].presetTime.allotted[7] := 1800.0;
   instHMISettings.instAniPNTmr.stations.me[32].presetTime.critical[7] := 300.0;
   instHMISettings.instAniPNTmr.stations.me[32].stackLightOut := 16#0400_0000;
   instHMISettings.instAniPNTmr.stations.me[33].dropZone := 3;
   instHMISettings.instAniPNTmr.stations.me[33].kp8Config.activate[7] := TRUE;
   instHMISettings.instAniPNTmr.stations.me[33].kp8Config.colorOn1[0] := 'off';
   instHMISettings.instAniPNTmr.stations.me[33].kp8Config.colorOn1[1] := 'off';
   instHMISettings.instAniPNTmr.stations.me[33].kp8Config.colorOn1[2] := 'off';
   instHMISettings.instAniPNTmr.stations.me[33].kp8Config.colorOn1[3] := 'off';
   instHMISettings.instAniPNTmr.stations.me[33].kp8Config.colorOn1[4] := 'off';
   instHMISettings.instAniPNTmr.stations.me[33].kp8Config.colorOn1[5] := 'off';
   instHMISettings.instAniPNTmr.stations.me[33].kp8Config.colorOn1[6] := 'off';
   instHMISettings.instAniPNTmr.stations.me[33].kp8Config.colorOn1[7] := 'yellow';
   instHMISettings.instAniPNTmr.stations.me[33].kp8Config.colorOn2[0] := 'off';
   instHMISettings.instAniPNTmr.stations.me[33].kp8Config.colorOn2[1] := 'off';
   instHMISettings.instAniPNTmr.stations.me[33].kp8Config.colorOn2[2] := 'off';
   instHMISettings.instAniPNTmr.stations.me[33].kp8Config.colorOn2[3] := 'off';
   instHMISettings.instAniPNTmr.stations.me[33].kp8Config.colorOn2[4] := 'off';
   instHMISettings.instAniPNTmr.stations.me[33].kp8Config.colorOn2[5] := 'off';
   instHMISettings.instAniPNTmr.stations.me[33].kp8Config.colorOn2[6] := 'off';
   instHMISettings.instAniPNTmr.stations.me[33].kp8Config.colorOff[0] := 'off';
   instHMISettings.instAniPNTmr.stations.me[33].kp8Config.colorOff[1] := 'off';
   instHMISettings.instAniPNTmr.stations.me[33].kp8Config.colorOff[2] := 'off';
   instHMISettings.instAniPNTmr.stations.me[33].kp8Config.colorOff[3] := 'off';
   instHMISettings.instAniPNTmr.stations.me[33].kp8Config.colorOff[4] := 'off';
   instHMISettings.instAniPNTmr.stations.me[33].kp8Config.colorOff[5] := 'off';
   instHMISettings.instAniPNTmr.stations.me[33].kp8Config.colorOff[6] := 'off';
   instHMISettings.instAniPNTmr.stations.me[33].kp8Config.colorOff[7] := 'green';
   instHMISettings.instAniPNTmr.stations.me[33].kp8Config.mode[7] := TRUE;
   instHMISettings.instAniPNTmr.stations.me[33].kp8Out := 16#0080_0000;
   instHMISettings.instAniPNTmr.stations.me[33].line := WSTRING#'1BX 2.0';
   instHMISettings.instAniPNTmr.stations.me[33].partNumbers[0] := WSTRING#'';
   instHMISettings.instAniPNTmr.stations.me[33].partNumbers[1] := WSTRING#'';
   instHMISettings.instAniPNTmr.stations.me[33].partNumbers[2] := WSTRING#'';
   instHMISettings.instAniPNTmr.stations.me[33].partNumbers[3] := WSTRING#'';
   instHMISettings.instAniPNTmr.stations.me[33].partNumbers[4] := WSTRING#'';
   instHMISettings.instAniPNTmr.stations.me[33].partNumbers[5] := WSTRING#'';
   instHMISettings.instAniPNTmr.stations.me[33].partNumbers[6] := WSTRING#'';
   instHMISettings.instAniPNTmr.stations.me[33].partNumbers[7] := WSTRING#'16.08.208.691.010D';
   instHMISettings.instAniPNTmr.stations.me[33].presetTime.allotted[7] := 1800.0;
   instHMISettings.instAniPNTmr.stations.me[33].presetTime.critical[7] := 300.0;
   instHMISettings.instAniPNTmr.stations.me[33].stackLightOut := 16#0400_0000;
   instHMISettings.instAniPNTmr.stations.me[34].dropZone := 4;
   instHMISettings.instAniPNTmr.stations.me[34].kp8Config.activate[3] := TRUE;
   instHMISettings.instAniPNTmr.stations.me[34].kp8Config.activate[7] := TRUE;
   instHMISettings.instAniPNTmr.stations.me[34].kp8Config.colorOn1[0] := 'off';
   instHMISettings.instAniPNTmr.stations.me[34].kp8Config.colorOn1[1] := 'off';
   instHMISettings.instAniPNTmr.stations.me[34].kp8Config.colorOn1[2] := 'off';
   instHMISettings.instAniPNTmr.stations.me[34].kp8Config.colorOn1[3] := 'yellow';
   instHMISettings.instAniPNTmr.stations.me[34].kp8Config.colorOn1[4] := 'off';
   instHMISettings.instAniPNTmr.stations.me[34].kp8Config.colorOn1[5] := 'off';
   instHMISettings.instAniPNTmr.stations.me[34].kp8Config.colorOn1[6] := 'off';
   instHMISettings.instAniPNTmr.stations.me[34].kp8Config.colorOn1[7] := 'yellow';
   instHMISettings.instAniPNTmr.stations.me[34].kp8Config.colorOn2[0] := 'off';
   instHMISettings.instAniPNTmr.stations.me[34].kp8Config.colorOn2[1] := 'off';
   instHMISettings.instAniPNTmr.stations.me[34].kp8Config.colorOn2[2] := 'off';
   instHMISettings.instAniPNTmr.stations.me[34].kp8Config.colorOn2[4] := 'off';
   instHMISettings.instAniPNTmr.stations.me[34].kp8Config.colorOn2[5] := 'off';
   instHMISettings.instAniPNTmr.stations.me[34].kp8Config.colorOn2[6] := 'off';
   instHMISettings.instAniPNTmr.stations.me[34].kp8Config.colorOff[0] := 'off';
   instHMISettings.instAniPNTmr.stations.me[34].kp8Config.colorOff[1] := 'off';
   instHMISettings.instAniPNTmr.stations.me[34].kp8Config.colorOff[2] := 'off';
   instHMISettings.instAniPNTmr.stations.me[34].kp8Config.colorOff[3] := 'green';
   instHMISettings.instAniPNTmr.stations.me[34].kp8Config.colorOff[4] := 'off';
   instHMISettings.instAniPNTmr.stations.me[34].kp8Config.colorOff[5] := 'off';
   instHMISettings.instAniPNTmr.stations.me[34].kp8Config.colorOff[6] := 'off';
   instHMISettings.instAniPNTmr.stations.me[34].kp8Config.colorOff[7] := 'green';
   instHMISettings.instAniPNTmr.stations.me[34].kp8Config.mode[3] := TRUE;
   instHMISettings.instAniPNTmr.stations.me[34].kp8Config.mode[7] := TRUE;
   instHMISettings.instAniPNTmr.stations.me[34].kp8Out := 16#0088_0000;
   instHMISettings.instAniPNTmr.stations.me[34].line := WSTRING#'1BX 2.0';
   instHMISettings.instAniPNTmr.stations.me[34].partNumbers[0] := WSTRING#'';
   instHMISettings.instAniPNTmr.stations.me[34].partNumbers[1] := WSTRING#'';
   instHMISettings.instAniPNTmr.stations.me[34].partNumbers[2] := WSTRING#'';
   instHMISettings.instAniPNTmr.stations.me[34].partNumbers[3] := WSTRING#'16.08.208.161.030E';
   instHMISettings.instAniPNTmr.stations.me[34].partNumbers[4] := WSTRING#'';
   instHMISettings.instAniPNTmr.stations.me[34].partNumbers[5] := WSTRING#'';
   instHMISettings.instAniPNTmr.stations.me[34].partNumbers[6] := WSTRING#'';
   instHMISettings.instAniPNTmr.stations.me[34].partNumbers[7] := WSTRING#'16.08.216.011.030B';
   instHMISettings.instAniPNTmr.stations.me[34].presetTime.allotted[3] := 1800.0;
   instHMISettings.instAniPNTmr.stations.me[34].presetTime.allotted[7] := 1800.0;
   instHMISettings.instAniPNTmr.stations.me[34].presetTime.critical[3] := 300.0;
   instHMISettings.instAniPNTmr.stations.me[34].presetTime.critical[7] := 300.0;
   instHMISettings.instAniPNTmr.stations.me[34].stackLightOut := 16#2400_0000;
   instHMISettings.instAniPNTmr.stations.me[35].dropZone := 5;
   instHMISettings.instAniPNTmr.stations.me[35].kp8Config.activate[3] := TRUE;
   instHMISettings.instAniPNTmr.stations.me[35].kp8Config.activate[7] := TRUE;
   instHMISettings.instAniPNTmr.stations.me[35].kp8Config.colorOn1[0] := 'off';
   instHMISettings.instAniPNTmr.stations.me[35].kp8Config.colorOn1[1] := 'off';
   instHMISettings.instAniPNTmr.stations.me[35].kp8Config.colorOn1[2] := 'off';
   instHMISettings.instAniPNTmr.stations.me[35].kp8Config.colorOn1[3] := 'yellow';
   instHMISettings.instAniPNTmr.stations.me[35].kp8Config.colorOn1[4] := 'off';
   instHMISettings.instAniPNTmr.stations.me[35].kp8Config.colorOn1[5] := 'off';
   instHMISettings.instAniPNTmr.stations.me[35].kp8Config.colorOn1[6] := 'off';
   instHMISettings.instAniPNTmr.stations.me[35].kp8Config.colorOn1[7] := 'yellow';
   instHMISettings.instAniPNTmr.stations.me[35].kp8Config.colorOn2[0] := 'off';
   instHMISettings.instAniPNTmr.stations.me[35].kp8Config.colorOn2[1] := 'off';
   instHMISettings.instAniPNTmr.stations.me[35].kp8Config.colorOn2[2] := 'off';
   instHMISettings.instAniPNTmr.stations.me[35].kp8Config.colorOn2[4] := 'off';
   instHMISettings.instAniPNTmr.stations.me[35].kp8Config.colorOn2[5] := 'off';
   instHMISettings.instAniPNTmr.stations.me[35].kp8Config.colorOn2[6] := 'off';
   instHMISettings.instAniPNTmr.stations.me[35].kp8Config.colorOff[0] := 'off';
   instHMISettings.instAniPNTmr.stations.me[35].kp8Config.colorOff[1] := 'off';
   instHMISettings.instAniPNTmr.stations.me[35].kp8Config.colorOff[2] := 'off';
   instHMISettings.instAniPNTmr.stations.me[35].kp8Config.colorOff[3] := 'green';
   instHMISettings.instAniPNTmr.stations.me[35].kp8Config.colorOff[4] := 'off';
   instHMISettings.instAniPNTmr.stations.me[35].kp8Config.colorOff[5] := 'off';
   instHMISettings.instAniPNTmr.stations.me[35].kp8Config.colorOff[6] := 'off';
   instHMISettings.instAniPNTmr.stations.me[35].kp8Config.colorOff[7] := 'green';
   instHMISettings.instAniPNTmr.stations.me[35].kp8Config.mode[3] := TRUE;
   instHMISettings.instAniPNTmr.stations.me[35].kp8Config.mode[7] := TRUE;
   instHMISettings.instAniPNTmr.stations.me[35].kp8Out := 16#0088_0000;
   instHMISettings.instAniPNTmr.stations.me[35].line := WSTRING#'1BX 2.0';
   instHMISettings.instAniPNTmr.stations.me[35].partNumbers[0] := WSTRING#'';
   instHMISettings.instAniPNTmr.stations.me[35].partNumbers[1] := WSTRING#'';
   instHMISettings.instAniPNTmr.stations.me[35].partNumbers[2] := WSTRING#'';
   instHMISettings.instAniPNTmr.stations.me[35].partNumbers[3] := WSTRING#'16.08.208.681.000K';
   instHMISettings.instAniPNTmr.stations.me[35].partNumbers[4] := WSTRING#'';
   instHMISettings.instAniPNTmr.stations.me[35].partNumbers[5] := WSTRING#'';
   instHMISettings.instAniPNTmr.stations.me[35].partNumbers[6] := WSTRING#'';
   instHMISettings.instAniPNTmr.stations.me[35].partNumbers[7] := WSTRING#'16.08.208.011.020I';
   instHMISettings.instAniPNTmr.stations.me[35].presetTime.allotted[3] := 1800.0;
   instHMISettings.instAniPNTmr.stations.me[35].presetTime.allotted[7] := 1800.0;
   instHMISettings.instAniPNTmr.stations.me[35].presetTime.critical[3] := 300.0;
   instHMISettings.instAniPNTmr.stations.me[35].presetTime.critical[7] := 300.0;
   instHMISettings.instAniPNTmr.stations.me[35].stackLightOut := 16#2400_0000;
   instHMISettings.instAniPNTmr.stations.me[36].dropZone := 1;
   instHMISettings.instAniPNTmr.stations.me[36].kp8Config.activate[3] := TRUE;
   instHMISettings.instAniPNTmr.stations.me[36].kp8Config.activate[7] := TRUE;
   instHMISettings.instAniPNTmr.stations.me[36].kp8Config.colorOn1[0] := 'off';
   instHMISettings.instAniPNTmr.stations.me[36].kp8Config.colorOn1[1] := 'off';
   instHMISettings.instAniPNTmr.stations.me[36].kp8Config.colorOn1[2] := 'off';
   instHMISettings.instAniPNTmr.stations.me[36].kp8Config.colorOn1[3] := 'yellow';
   instHMISettings.instAniPNTmr.stations.me[36].kp8Config.colorOn1[4] := 'off';
   instHMISettings.instAniPNTmr.stations.me[36].kp8Config.colorOn1[5] := 'off';
   instHMISettings.instAniPNTmr.stations.me[36].kp8Config.colorOn1[6] := 'off';
   instHMISettings.instAniPNTmr.stations.me[36].kp8Config.colorOn1[7] := 'yellow';
   instHMISettings.instAniPNTmr.stations.me[36].kp8Config.colorOn2[0] := 'off';
   instHMISettings.instAniPNTmr.stations.me[36].kp8Config.colorOn2[1] := 'off';
   instHMISettings.instAniPNTmr.stations.me[36].kp8Config.colorOn2[2] := 'off';
   instHMISettings.instAniPNTmr.stations.me[36].kp8Config.colorOn2[4] := 'off';
   instHMISettings.instAniPNTmr.stations.me[36].kp8Config.colorOn2[5] := 'off';
   instHMISettings.instAniPNTmr.stations.me[36].kp8Config.colorOn2[6] := 'off';
   instHMISettings.instAniPNTmr.stations.me[36].kp8Config.colorOff[0] := 'off';
   instHMISettings.instAniPNTmr.stations.me[36].kp8Config.colorOff[1] := 'off';
   instHMISettings.instAniPNTmr.stations.me[36].kp8Config.colorOff[2] := 'off';
   instHMISettings.instAniPNTmr.stations.me[36].kp8Config.colorOff[3] := 'green';
   instHMISettings.instAniPNTmr.stations.me[36].kp8Config.colorOff[4] := 'off';
   instHMISettings.instAniPNTmr.stations.me[36].kp8Config.colorOff[5] := 'off';
   instHMISettings.instAniPNTmr.stations.me[36].kp8Config.colorOff[6] := 'off';
   instHMISettings.instAniPNTmr.stations.me[36].kp8Config.colorOff[7] := 'green';
   instHMISettings.instAniPNTmr.stations.me[36].kp8Config.mode[3] := TRUE;
   instHMISettings.instAniPNTmr.stations.me[36].kp8Config.mode[7] := TRUE;
   instHMISettings.instAniPNTmr.stations.me[36].kp8Out := 16#0088_0000;
   instHMISettings.instAniPNTmr.stations.me[36].line := WSTRING#'1BX 3.0';
   instHMISettings.instAniPNTmr.stations.me[36].partNumbers[0] := WSTRING#'';
   instHMISettings.instAniPNTmr.stations.me[36].partNumbers[1] := WSTRING#'';
   instHMISettings.instAniPNTmr.stations.me[36].partNumbers[2] := WSTRING#'';
   instHMISettings.instAniPNTmr.stations.me[36].partNumbers[3] := WSTRING#'16.08.208.011.020I';
   instHMISettings.instAniPNTmr.stations.me[36].partNumbers[4] := WSTRING#'';
   instHMISettings.instAniPNTmr.stations.me[36].partNumbers[5] := WSTRING#'';
   instHMISettings.instAniPNTmr.stations.me[36].partNumbers[6] := WSTRING#'';
   instHMISettings.instAniPNTmr.stations.me[36].partNumbers[7] := WSTRING#'16.08.208.681.000K';
   instHMISettings.instAniPNTmr.stations.me[36].presetTime.allotted[3] := 1800.0;
   instHMISettings.instAniPNTmr.stations.me[36].presetTime.allotted[7] := 1800.0;
   instHMISettings.instAniPNTmr.stations.me[36].presetTime.critical[3] := 300.0;
   instHMISettings.instAniPNTmr.stations.me[36].presetTime.critical[7] := 300.0;
   instHMISettings.instAniPNTmr.stations.me[36].stackLightOut := 16#2400_0000;
   instHMISettings.instAniPNTmr.stations.me[37].dropZone := 2;
   instHMISettings.instAniPNTmr.stations.me[37].kp8Config.activate[3] := TRUE;
   instHMISettings.instAniPNTmr.stations.me[37].kp8Config.activate[7] := TRUE;
   instHMISettings.instAniPNTmr.stations.me[37].kp8Config.colorOn1[0] := 'off';
   instHMISettings.instAniPNTmr.stations.me[37].kp8Config.colorOn1[1] := 'off';
   instHMISettings.instAniPNTmr.stations.me[37].kp8Config.colorOn1[2] := 'off';
   instHMISettings.instAniPNTmr.stations.me[37].kp8Config.colorOn1[3] := 'yellow';
   instHMISettings.instAniPNTmr.stations.me[37].kp8Config.colorOn1[4] := 'off';
   instHMISettings.instAniPNTmr.stations.me[37].kp8Config.colorOn1[5] := 'off';
   instHMISettings.instAniPNTmr.stations.me[37].kp8Config.colorOn1[6] := 'off';
   instHMISettings.instAniPNTmr.stations.me[37].kp8Config.colorOn1[7] := 'yellow';
   instHMISettings.instAniPNTmr.stations.me[37].kp8Config.colorOn2[0] := 'off';
   instHMISettings.instAniPNTmr.stations.me[37].kp8Config.colorOn2[1] := 'off';
   instHMISettings.instAniPNTmr.stations.me[37].kp8Config.colorOn2[2] := 'off';
   instHMISettings.instAniPNTmr.stations.me[37].kp8Config.colorOn2[4] := 'off';
   instHMISettings.instAniPNTmr.stations.me[37].kp8Config.colorOn2[5] := 'off';
   instHMISettings.instAniPNTmr.stations.me[37].kp8Config.colorOn2[6] := 'off';
   instHMISettings.instAniPNTmr.stations.me[37].kp8Config.colorOff[0] := 'off';
   instHMISettings.instAniPNTmr.stations.me[37].kp8Config.colorOff[1] := 'off';
   instHMISettings.instAniPNTmr.stations.me[37].kp8Config.colorOff[2] := 'off';
   instHMISettings.instAniPNTmr.stations.me[37].kp8Config.colorOff[3] := 'green';
   instHMISettings.instAniPNTmr.stations.me[37].kp8Config.colorOff[4] := 'off';
   instHMISettings.instAniPNTmr.stations.me[37].kp8Config.colorOff[5] := 'off';
   instHMISettings.instAniPNTmr.stations.me[37].kp8Config.colorOff[6] := 'off';
   instHMISettings.instAniPNTmr.stations.me[37].kp8Config.colorOff[7] := 'green';
   instHMISettings.instAniPNTmr.stations.me[37].kp8Config.mode[3] := TRUE;
   instHMISettings.instAniPNTmr.stations.me[37].kp8Config.mode[7] := TRUE;
   instHMISettings.instAniPNTmr.stations.me[37].kp8Out := 16#0088_0000;
   instHMISettings.instAniPNTmr.stations.me[37].line := WSTRING#'1BX 3.0';
   instHMISettings.instAniPNTmr.stations.me[37].partNumbers[0] := WSTRING#'';
   instHMISettings.instAniPNTmr.stations.me[37].partNumbers[1] := WSTRING#'';
   instHMISettings.instAniPNTmr.stations.me[37].partNumbers[2] := WSTRING#'';
   instHMISettings.instAniPNTmr.stations.me[37].partNumbers[3] := WSTRING#'16.08.216.011.030B';
   instHMISettings.instAniPNTmr.stations.me[37].partNumbers[4] := WSTRING#'';
   instHMISettings.instAniPNTmr.stations.me[37].partNumbers[5] := WSTRING#'';
   instHMISettings.instAniPNTmr.stations.me[37].partNumbers[6] := WSTRING#'';
   instHMISettings.instAniPNTmr.stations.me[37].partNumbers[7] := WSTRING#'16.08.208.161.030E';
   instHMISettings.instAniPNTmr.stations.me[37].presetTime.allotted[3] := 1800.0;
   instHMISettings.instAniPNTmr.stations.me[37].presetTime.allotted[7] := 1800.0;
   instHMISettings.instAniPNTmr.stations.me[37].presetTime.critical[3] := 300.0;
   instHMISettings.instAniPNTmr.stations.me[37].presetTime.critical[7] := 300.0;
   instHMISettings.instAniPNTmr.stations.me[37].stackLightOut := 16#2400_0000;
   instHMISettings.instAniPNTmr.stations.me[38].dropZone := 3;
   instHMISettings.instAniPNTmr.stations.me[38].kp8Config.activate[7] := TRUE;
   instHMISettings.instAniPNTmr.stations.me[38].kp8Config.colorOn1[0] := 'off';
   instHMISettings.instAniPNTmr.stations.me[38].kp8Config.colorOn1[1] := 'off';
   instHMISettings.instAniPNTmr.stations.me[38].kp8Config.colorOn1[2] := 'off';
   instHMISettings.instAniPNTmr.stations.me[38].kp8Config.colorOn1[3] := 'off';
   instHMISettings.instAniPNTmr.stations.me[38].kp8Config.colorOn1[4] := 'off';
   instHMISettings.instAniPNTmr.stations.me[38].kp8Config.colorOn1[5] := 'off';
   instHMISettings.instAniPNTmr.stations.me[38].kp8Config.colorOn1[6] := 'off';
   instHMISettings.instAniPNTmr.stations.me[38].kp8Config.colorOn1[7] := 'yellow';
   instHMISettings.instAniPNTmr.stations.me[38].kp8Config.colorOn2[0] := 'off';
   instHMISettings.instAniPNTmr.stations.me[38].kp8Config.colorOn2[1] := 'off';
   instHMISettings.instAniPNTmr.stations.me[38].kp8Config.colorOn2[2] := 'off';
   instHMISettings.instAniPNTmr.stations.me[38].kp8Config.colorOn2[3] := 'off';
   instHMISettings.instAniPNTmr.stations.me[38].kp8Config.colorOn2[4] := 'off';
   instHMISettings.instAniPNTmr.stations.me[38].kp8Config.colorOn2[5] := 'off';
   instHMISettings.instAniPNTmr.stations.me[38].kp8Config.colorOn2[6] := 'off';
   instHMISettings.instAniPNTmr.stations.me[38].kp8Config.colorOff[0] := 'off';
   instHMISettings.instAniPNTmr.stations.me[38].kp8Config.colorOff[1] := 'off';
   instHMISettings.instAniPNTmr.stations.me[38].kp8Config.colorOff[2] := 'off';
   instHMISettings.instAniPNTmr.stations.me[38].kp8Config.colorOff[3] := 'off';
   instHMISettings.instAniPNTmr.stations.me[38].kp8Config.colorOff[4] := 'off';
   instHMISettings.instAniPNTmr.stations.me[38].kp8Config.colorOff[5] := 'off';
   instHMISettings.instAniPNTmr.stations.me[38].kp8Config.colorOff[6] := 'off';
   instHMISettings.instAniPNTmr.stations.me[38].kp8Config.colorOff[7] := 'green';
   instHMISettings.instAniPNTmr.stations.me[38].kp8Config.mode[7] := TRUE;
   instHMISettings.instAniPNTmr.stations.me[38].kp8Out := 16#0080_0000;
   instHMISettings.instAniPNTmr.stations.me[38].line := WSTRING#'1BX 3.0';
   instHMISettings.instAniPNTmr.stations.me[38].partNumbers[0] := WSTRING#'';
   instHMISettings.instAniPNTmr.stations.me[38].partNumbers[1] := WSTRING#'';
   instHMISettings.instAniPNTmr.stations.me[38].partNumbers[2] := WSTRING#'';
   instHMISettings.instAniPNTmr.stations.me[38].partNumbers[3] := WSTRING#'';
   instHMISettings.instAniPNTmr.stations.me[38].partNumbers[4] := WSTRING#'';
   instHMISettings.instAniPNTmr.stations.me[38].partNumbers[5] := WSTRING#'';
   instHMISettings.instAniPNTmr.stations.me[38].partNumbers[6] := WSTRING#'';
   instHMISettings.instAniPNTmr.stations.me[38].partNumbers[7] := WSTRING#'16.08.208.601.010D';
   instHMISettings.instAniPNTmr.stations.me[38].presetTime.allotted[7] := 1800.0;
   instHMISettings.instAniPNTmr.stations.me[38].presetTime.critical[7] := 300.0;
   instHMISettings.instAniPNTmr.stations.me[38].stackLightOut := 16#0400_0000;
   instHMISettings.instAniPNTmr.instPNEntEnable.disable := TRUE;
   instHMISettings.instAniPNTmr.instPNEntEnable.assignAnimate := 254;
   instHMISettings.instAniPNTmr.instPNEntEnable.ioFieldAnimate := 254;
   instHMISettings.instAniPNTmr.instAlltEntEnable.disable := TRUE;
   instHMISettings.instAniPNTmr.instAlltEntEnable.assignAnimate := 254;
   instHMISettings.instAniPNTmr.instAlltEntEnable.ioFieldAnimate := 254;
   instHMISettings.instAniPNTmr.instCrtEntEnable.disable := TRUE;
   instHMISettings.instAniPNTmr.instCrtEntEnable.assignAnimate := 254;
   instHMISettings.instAniPNTmr.instCrtEntEnable.ioFieldAnimate := 254;
   instInitialize.rtElapsed := 0.00503095;
   instInitialize.rt.elapsed := 0.00503095;
   instInitialize.rt.mem := 1.03108171604573E-306;
   instKP8BtnAct.old.kp8Config[0].activate[3] := TRUE;
   instKP8BtnAct.old.kp8Config[0].activate[7] := TRUE;
   instKP8BtnAct.old.kp8Config[0].colorOn1[0] := 'off';
   instKP8BtnAct.old.kp8Config[0].colorOn1[1] := 'off';
   instKP8BtnAct.old.kp8Config[0].colorOn1[2] := 'off';
   instKP8BtnAct.old.kp8Config[0].colorOn1[3] := 'yellow';
   instKP8BtnAct.old.kp8Config[0].colorOn1[4] := 'off';
   instKP8BtnAct.old.kp8Config[0].colorOn1[5] := 'off';
   instKP8BtnAct.old.kp8Config[0].colorOn1[6] := 'off';
   instKP8BtnAct.old.kp8Config[0].colorOn1[7] := 'yellow';
   instKP8BtnAct.old.kp8Config[0].colorOn2[0] := 'off';
   instKP8BtnAct.old.kp8Config[0].colorOn2[1] := 'off';
   instKP8BtnAct.old.kp8Config[0].colorOn2[2] := 'off';
   instKP8BtnAct.old.kp8Config[0].colorOn2[4] := 'off';
   instKP8BtnAct.old.kp8Config[0].colorOn2[5] := 'off';
   instKP8BtnAct.old.kp8Config[0].colorOn2[6] := 'off';
   instKP8BtnAct.old.kp8Config[0].colorOff[0] := 'off';
   instKP8BtnAct.old.kp8Config[0].colorOff[1] := 'off';
   instKP8BtnAct.old.kp8Config[0].colorOff[2] := 'off';
   instKP8BtnAct.old.kp8Config[0].colorOff[3] := 'green';
   instKP8BtnAct.old.kp8Config[0].colorOff[4] := 'off';
   instKP8BtnAct.old.kp8Config[0].colorOff[5] := 'off';
   instKP8BtnAct.old.kp8Config[0].colorOff[6] := 'off';
   instKP8BtnAct.old.kp8Config[0].colorOff[7] := 'green';
   instKP8BtnAct.old.kp8Config[0].mode[3] := TRUE;
   instKP8BtnAct.old.kp8Config[0].mode[7] := TRUE;
   instKP8BtnAct.old.kp8Config[1].activate[2] := TRUE;
   instKP8BtnAct.old.kp8Config[1].activate[3] := TRUE;
   instKP8BtnAct.old.kp8Config[1].activate[6] := TRUE;
   instKP8BtnAct.old.kp8Config[1].activate[7] := TRUE;
   instKP8BtnAct.old.kp8Config[1].colorOn1[0] := 'off';
   instKP8BtnAct.old.kp8Config[1].colorOn1[1] := 'off';
   instKP8BtnAct.old.kp8Config[1].colorOn1[2] := 'yellow';
   instKP8BtnAct.old.kp8Config[1].colorOn1[3] := 'yellow';
   instKP8BtnAct.old.kp8Config[1].colorOn1[4] := 'off';
   instKP8BtnAct.old.kp8Config[1].colorOn1[5] := 'off';
   instKP8BtnAct.old.kp8Config[1].colorOn1[6] := 'yellow';
   instKP8BtnAct.old.kp8Config[1].colorOn1[7] := 'yellow';
   instKP8BtnAct.old.kp8Config[1].colorOn2[0] := 'off';
   instKP8BtnAct.old.kp8Config[1].colorOn2[1] := 'off';
   instKP8BtnAct.old.kp8Config[1].colorOn2[4] := 'off';
   instKP8BtnAct.old.kp8Config[1].colorOn2[5] := 'off';
   instKP8BtnAct.old.kp8Config[1].colorOff[0] := 'off';
   instKP8BtnAct.old.kp8Config[1].colorOff[1] := 'off';
   instKP8BtnAct.old.kp8Config[1].colorOff[2] := 'green';
   instKP8BtnAct.old.kp8Config[1].colorOff[3] := 'green';
   instKP8BtnAct.old.kp8Config[1].colorOff[4] := 'off';
   instKP8BtnAct.old.kp8Config[1].colorOff[5] := 'off';
   instKP8BtnAct.old.kp8Config[1].colorOff[6] := 'green';
   instKP8BtnAct.old.kp8Config[1].colorOff[7] := 'green';
   instKP8BtnAct.old.kp8Config[1].mode[2] := TRUE;
   instKP8BtnAct.old.kp8Config[1].mode[3] := TRUE;
   instKP8BtnAct.old.kp8Config[1].mode[6] := TRUE;
   instKP8BtnAct.old.kp8Config[1].mode[7] := TRUE;
   instKP8BtnAct.old.kp8Config[2].activate[1] := TRUE;
   instKP8BtnAct.old.kp8Config[2].activate[2] := TRUE;
   instKP8BtnAct.old.kp8Config[2].activate[3] := TRUE;
   instKP8BtnAct.old.kp8Config[2].activate[5] := TRUE;
   instKP8BtnAct.old.kp8Config[2].activate[6] := TRUE;
   instKP8BtnAct.old.kp8Config[2].activate[7] := TRUE;
   instKP8BtnAct.old.kp8Config[2].colorOn1[0] := 'off';
   instKP8BtnAct.old.kp8Config[2].colorOn1[1] := 'yellow';
   instKP8BtnAct.old.kp8Config[2].colorOn1[2] := 'yellow';
   instKP8BtnAct.old.kp8Config[2].colorOn1[3] := 'yellow';
   instKP8BtnAct.old.kp8Config[2].colorOn1[4] := 'off';
   instKP8BtnAct.old.kp8Config[2].colorOn1[5] := 'yellow';
   instKP8BtnAct.old.kp8Config[2].colorOn1[6] := 'yellow';
   instKP8BtnAct.old.kp8Config[2].colorOn1[7] := 'yellow';
   instKP8BtnAct.old.kp8Config[2].colorOn2[0] := 'off';
   instKP8BtnAct.old.kp8Config[2].colorOn2[4] := 'off';
   instKP8BtnAct.old.kp8Config[2].colorOff[0] := 'off';
   instKP8BtnAct.old.kp8Config[2].colorOff[1] := 'green';
   instKP8BtnAct.old.kp8Config[2].colorOff[2] := 'green';
   instKP8BtnAct.old.kp8Config[2].colorOff[3] := 'green';
   instKP8BtnAct.old.kp8Config[2].colorOff[4] := 'off';
   instKP8BtnAct.old.kp8Config[2].colorOff[5] := 'green';
   instKP8BtnAct.old.kp8Config[2].colorOff[6] := 'green';
   instKP8BtnAct.old.kp8Config[2].colorOff[7] := 'green';
   instKP8BtnAct.old.kp8Config[2].mode[1] := TRUE;
   instKP8BtnAct.old.kp8Config[2].mode[2] := TRUE;
   instKP8BtnAct.old.kp8Config[2].mode[3] := TRUE;
   instKP8BtnAct.old.kp8Config[2].mode[5] := TRUE;
   instKP8BtnAct.old.kp8Config[2].mode[6] := TRUE;
   instKP8BtnAct.old.kp8Config[2].mode[7] := TRUE;
   instKP8BtnAct.old.kp8Config[3].activate[1] := TRUE;
   instKP8BtnAct.old.kp8Config[3].activate[2] := TRUE;
   instKP8BtnAct.old.kp8Config[3].activate[3] := TRUE;
   instKP8BtnAct.old.kp8Config[3].activate[5] := TRUE;
   instKP8BtnAct.old.kp8Config[3].activate[6] := TRUE;
   instKP8BtnAct.old.kp8Config[3].activate[7] := TRUE;
   instKP8BtnAct.old.kp8Config[3].colorOn1[0] := 'off';
   instKP8BtnAct.old.kp8Config[3].colorOn1[1] := 'yellow';
   instKP8BtnAct.old.kp8Config[3].colorOn1[2] := 'yellow';
   instKP8BtnAct.old.kp8Config[3].colorOn1[3] := 'yellow';
   instKP8BtnAct.old.kp8Config[3].colorOn1[4] := 'off';
   instKP8BtnAct.old.kp8Config[3].colorOn1[5] := 'yellow';
   instKP8BtnAct.old.kp8Config[3].colorOn1[6] := 'yellow';
   instKP8BtnAct.old.kp8Config[3].colorOn1[7] := 'yellow';
   instKP8BtnAct.old.kp8Config[3].colorOn2[0] := 'off';
   instKP8BtnAct.old.kp8Config[3].colorOn2[4] := 'off';
   instKP8BtnAct.old.kp8Config[3].colorOff[0] := 'off';
   instKP8BtnAct.old.kp8Config[3].colorOff[1] := 'green';
   instKP8BtnAct.old.kp8Config[3].colorOff[2] := 'green';
   instKP8BtnAct.old.kp8Config[3].colorOff[3] := 'green';
   instKP8BtnAct.old.kp8Config[3].colorOff[4] := 'off';
   instKP8BtnAct.old.kp8Config[3].colorOff[5] := 'green';
   instKP8BtnAct.old.kp8Config[3].colorOff[6] := 'green';
   instKP8BtnAct.old.kp8Config[3].colorOff[7] := 'green';
   instKP8BtnAct.old.kp8Config[3].mode[1] := TRUE;
   instKP8BtnAct.old.kp8Config[3].mode[2] := TRUE;
   instKP8BtnAct.old.kp8Config[3].mode[3] := TRUE;
   instKP8BtnAct.old.kp8Config[3].mode[5] := TRUE;
   instKP8BtnAct.old.kp8Config[3].mode[6] := TRUE;
   instKP8BtnAct.old.kp8Config[3].mode[7] := TRUE;
   instKP8BtnAct.old.kp8Config[4].activate[7] := TRUE;
   instKP8BtnAct.old.kp8Config[4].colorOn1[0] := 'off';
   instKP8BtnAct.old.kp8Config[4].colorOn1[1] := 'off';
   instKP8BtnAct.old.kp8Config[4].colorOn1[2] := 'off';
   instKP8BtnAct.old.kp8Config[4].colorOn1[3] := 'off';
   instKP8BtnAct.old.kp8Config[4].colorOn1[4] := 'off';
   instKP8BtnAct.old.kp8Config[4].colorOn1[5] := 'off';
   instKP8BtnAct.old.kp8Config[4].colorOn1[6] := 'off';
   instKP8BtnAct.old.kp8Config[4].colorOn1[7] := 'yellow';
   instKP8BtnAct.old.kp8Config[4].colorOn2[0] := 'off';
   instKP8BtnAct.old.kp8Config[4].colorOn2[1] := 'off';
   instKP8BtnAct.old.kp8Config[4].colorOn2[2] := 'off';
   instKP8BtnAct.old.kp8Config[4].colorOn2[3] := 'off';
   instKP8BtnAct.old.kp8Config[4].colorOn2[4] := 'off';
   instKP8BtnAct.old.kp8Config[4].colorOn2[5] := 'off';
   instKP8BtnAct.old.kp8Config[4].colorOn2[6] := 'off';
   instKP8BtnAct.old.kp8Config[4].colorOff[0] := 'off';
   instKP8BtnAct.old.kp8Config[4].colorOff[1] := 'off';
   instKP8BtnAct.old.kp8Config[4].colorOff[2] := 'off';
   instKP8BtnAct.old.kp8Config[4].colorOff[3] := 'off';
   instKP8BtnAct.old.kp8Config[4].colorOff[4] := 'off';
   instKP8BtnAct.old.kp8Config[4].colorOff[5] := 'off';
   instKP8BtnAct.old.kp8Config[4].colorOff[6] := 'off';
   instKP8BtnAct.old.kp8Config[4].colorOff[7] := 'green';
   instKP8BtnAct.old.kp8Config[4].mode[7] := TRUE;
   instKP8BtnAct.old.kp8Config[5].activate[1] := TRUE;
   instKP8BtnAct.old.kp8Config[5].activate[2] := TRUE;
   instKP8BtnAct.old.kp8Config[5].activate[3] := TRUE;
   instKP8BtnAct.old.kp8Config[5].activate[5] := TRUE;
   instKP8BtnAct.old.kp8Config[5].activate[6] := TRUE;
   instKP8BtnAct.old.kp8Config[5].activate[7] := TRUE;
   instKP8BtnAct.old.kp8Config[5].colorOn1[0] := 'off';
   instKP8BtnAct.old.kp8Config[5].colorOn1[1] := 'yellow';
   instKP8BtnAct.old.kp8Config[5].colorOn1[2] := 'yellow';
   instKP8BtnAct.old.kp8Config[5].colorOn1[3] := 'yellow';
   instKP8BtnAct.old.kp8Config[5].colorOn1[4] := 'off';
   instKP8BtnAct.old.kp8Config[5].colorOn1[5] := 'yellow';
   instKP8BtnAct.old.kp8Config[5].colorOn1[6] := 'yellow';
   instKP8BtnAct.old.kp8Config[5].colorOn1[7] := 'yellow';
   instKP8BtnAct.old.kp8Config[5].colorOn2[0] := 'off';
   instKP8BtnAct.old.kp8Config[5].colorOn2[4] := 'off';
   instKP8BtnAct.old.kp8Config[5].colorOff[0] := 'off';
   instKP8BtnAct.old.kp8Config[5].colorOff[1] := 'green';
   instKP8BtnAct.old.kp8Config[5].colorOff[2] := 'green';
   instKP8BtnAct.old.kp8Config[5].colorOff[3] := 'green';
   instKP8BtnAct.old.kp8Config[5].colorOff[4] := 'off';
   instKP8BtnAct.old.kp8Config[5].colorOff[5] := 'green';
   instKP8BtnAct.old.kp8Config[5].colorOff[6] := 'green';
   instKP8BtnAct.old.kp8Config[5].colorOff[7] := 'green';
   instKP8BtnAct.old.kp8Config[5].mode[1] := TRUE;
   instKP8BtnAct.old.kp8Config[5].mode[2] := TRUE;
   instKP8BtnAct.old.kp8Config[5].mode[3] := TRUE;
   instKP8BtnAct.old.kp8Config[5].mode[5] := TRUE;
   instKP8BtnAct.old.kp8Config[5].mode[6] := TRUE;
   instKP8BtnAct.old.kp8Config[5].mode[7] := TRUE;
   instKP8BtnAct.old.kp8Config[6].activate[1] := TRUE;
   instKP8BtnAct.old.kp8Config[6].activate[2] := TRUE;
   instKP8BtnAct.old.kp8Config[6].activate[3] := TRUE;
   instKP8BtnAct.old.kp8Config[6].activate[5] := TRUE;
   instKP8BtnAct.old.kp8Config[6].activate[6] := TRUE;
   instKP8BtnAct.old.kp8Config[6].activate[7] := TRUE;
   instKP8BtnAct.old.kp8Config[6].colorOn1[0] := 'off';
   instKP8BtnAct.old.kp8Config[6].colorOn1[1] := 'yellow';
   instKP8BtnAct.old.kp8Config[6].colorOn1[2] := 'yellow';
   instKP8BtnAct.old.kp8Config[6].colorOn1[3] := 'yellow';
   instKP8BtnAct.old.kp8Config[6].colorOn1[4] := 'off';
   instKP8BtnAct.old.kp8Config[6].colorOn1[5] := 'yellow';
   instKP8BtnAct.old.kp8Config[6].colorOn1[6] := 'yellow';
   instKP8BtnAct.old.kp8Config[6].colorOn1[7] := 'yellow';
   instKP8BtnAct.old.kp8Config[6].colorOn2[0] := 'off';
   instKP8BtnAct.old.kp8Config[6].colorOn2[4] := 'off';
   instKP8BtnAct.old.kp8Config[6].colorOff[0] := 'off';
   instKP8BtnAct.old.kp8Config[6].colorOff[1] := 'green';
   instKP8BtnAct.old.kp8Config[6].colorOff[2] := 'green';
   instKP8BtnAct.old.kp8Config[6].colorOff[3] := 'green';
   instKP8BtnAct.old.kp8Config[6].colorOff[4] := 'off';
   instKP8BtnAct.old.kp8Config[6].colorOff[5] := 'green';
   instKP8BtnAct.old.kp8Config[6].colorOff[6] := 'green';
   instKP8BtnAct.old.kp8Config[6].colorOff[7] := 'green';
   instKP8BtnAct.old.kp8Config[6].mode[1] := TRUE;
   instKP8BtnAct.old.kp8Config[6].mode[2] := TRUE;
   instKP8BtnAct.old.kp8Config[6].mode[3] := TRUE;
   instKP8BtnAct.old.kp8Config[6].mode[5] := TRUE;
   instKP8BtnAct.old.kp8Config[6].mode[6] := TRUE;
   instKP8BtnAct.old.kp8Config[6].mode[7] := TRUE;
   instKP8BtnAct.old.kp8Config[7].activate[3] := TRUE;
   instKP8BtnAct.old.kp8Config[7].activate[6] := TRUE;
   instKP8BtnAct.old.kp8Config[7].activate[7] := TRUE;
   instKP8BtnAct.old.kp8Config[7].colorOn1[0] := 'off';
   instKP8BtnAct.old.kp8Config[7].colorOn1[1] := 'off';
   instKP8BtnAct.old.kp8Config[7].colorOn1[2] := 'off';
   instKP8BtnAct.old.kp8Config[7].colorOn1[3] := 'yellow';
   instKP8BtnAct.old.kp8Config[7].colorOn1[4] := 'off';
   instKP8BtnAct.old.kp8Config[7].colorOn1[5] := 'off';
   instKP8BtnAct.old.kp8Config[7].colorOn1[6] := 'yellow';
   instKP8BtnAct.old.kp8Config[7].colorOn1[7] := 'yellow';
   instKP8BtnAct.old.kp8Config[7].colorOn2[0] := 'off';
   instKP8BtnAct.old.kp8Config[7].colorOn2[1] := 'off';
   instKP8BtnAct.old.kp8Config[7].colorOn2[2] := 'off';
   instKP8BtnAct.old.kp8Config[7].colorOn2[4] := 'off';
   instKP8BtnAct.old.kp8Config[7].colorOn2[5] := 'off';
   instKP8BtnAct.old.kp8Config[7].colorOff[0] := 'off';
   instKP8BtnAct.old.kp8Config[7].colorOff[1] := 'off';
   instKP8BtnAct.old.kp8Config[7].colorOff[2] := 'off';
   instKP8BtnAct.old.kp8Config[7].colorOff[3] := 'green';
   instKP8BtnAct.old.kp8Config[7].colorOff[4] := 'off';
   instKP8BtnAct.old.kp8Config[7].colorOff[5] := 'off';
   instKP8BtnAct.old.kp8Config[7].colorOff[6] := 'green';
   instKP8BtnAct.old.kp8Config[7].colorOff[7] := 'green';
   instKP8BtnAct.old.kp8Config[7].mode[3] := TRUE;
   instKP8BtnAct.old.kp8Config[7].mode[6] := TRUE;
   instKP8BtnAct.old.kp8Config[7].mode[7] := TRUE;
   instKP8BtnAct.old.kp8Config[8].activate[3] := TRUE;
   instKP8BtnAct.old.kp8Config[8].activate[6] := TRUE;
   instKP8BtnAct.old.kp8Config[8].activate[7] := TRUE;
   instKP8BtnAct.old.kp8Config[8].colorOn1[0] := 'off';
   instKP8BtnAct.old.kp8Config[8].colorOn1[1] := 'off';
   instKP8BtnAct.old.kp8Config[8].colorOn1[2] := 'off';
   instKP8BtnAct.old.kp8Config[8].colorOn1[3] := 'yellow';
   instKP8BtnAct.old.kp8Config[8].colorOn1[4] := 'off';
   instKP8BtnAct.old.kp8Config[8].colorOn1[5] := 'off';
   instKP8BtnAct.old.kp8Config[8].colorOn1[6] := 'yellow';
   instKP8BtnAct.old.kp8Config[8].colorOn1[7] := 'yellow';
   instKP8BtnAct.old.kp8Config[8].colorOn2[0] := 'off';
   instKP8BtnAct.old.kp8Config[8].colorOn2[1] := 'off';
   instKP8BtnAct.old.kp8Config[8].colorOn2[2] := 'off';
   instKP8BtnAct.old.kp8Config[8].colorOn2[4] := 'off';
   instKP8BtnAct.old.kp8Config[8].colorOn2[5] := 'off';
   instKP8BtnAct.old.kp8Config[8].colorOff[0] := 'off';
   instKP8BtnAct.old.kp8Config[8].colorOff[1] := 'off';
   instKP8BtnAct.old.kp8Config[8].colorOff[2] := 'off';
   instKP8BtnAct.old.kp8Config[8].colorOff[3] := 'green';
   instKP8BtnAct.old.kp8Config[8].colorOff[4] := 'off';
   instKP8BtnAct.old.kp8Config[8].colorOff[5] := 'off';
   instKP8BtnAct.old.kp8Config[8].colorOff[6] := 'green';
   instKP8BtnAct.old.kp8Config[8].colorOff[7] := 'green';
   instKP8BtnAct.old.kp8Config[8].mode[3] := TRUE;
   instKP8BtnAct.old.kp8Config[8].mode[6] := TRUE;
   instKP8BtnAct.old.kp8Config[8].mode[7] := TRUE;
   instKP8BtnAct.old.kp8Config[9].activate[3] := TRUE;
   instKP8BtnAct.old.kp8Config[9].activate[7] := TRUE;
   instKP8BtnAct.old.kp8Config[9].colorOn1[0] := 'off';
   instKP8BtnAct.old.kp8Config[9].colorOn1[1] := 'off';
   instKP8BtnAct.old.kp8Config[9].colorOn1[2] := 'off';
   instKP8BtnAct.old.kp8Config[9].colorOn1[3] := 'yellow';
   instKP8BtnAct.old.kp8Config[9].colorOn1[4] := 'off';
   instKP8BtnAct.old.kp8Config[9].colorOn1[5] := 'off';
   instKP8BtnAct.old.kp8Config[9].colorOn1[6] := 'off';
   instKP8BtnAct.old.kp8Config[9].colorOn1[7] := 'yellow';
   instKP8BtnAct.old.kp8Config[9].colorOn2[0] := 'off';
   instKP8BtnAct.old.kp8Config[9].colorOn2[1] := 'off';
   instKP8BtnAct.old.kp8Config[9].colorOn2[2] := 'off';
   instKP8BtnAct.old.kp8Config[9].colorOn2[4] := 'off';
   instKP8BtnAct.old.kp8Config[9].colorOn2[5] := 'off';
   instKP8BtnAct.old.kp8Config[9].colorOn2[6] := 'off';
   instKP8BtnAct.old.kp8Config[9].colorOff[0] := 'off';
   instKP8BtnAct.old.kp8Config[9].colorOff[1] := 'off';
   instKP8BtnAct.old.kp8Config[9].colorOff[2] := 'off';
   instKP8BtnAct.old.kp8Config[9].colorOff[3] := 'green';
   instKP8BtnAct.old.kp8Config[9].colorOff[4] := 'off';
   instKP8BtnAct.old.kp8Config[9].colorOff[5] := 'off';
   instKP8BtnAct.old.kp8Config[9].colorOff[6] := 'off';
   instKP8BtnAct.old.kp8Config[9].colorOff[7] := 'green';
   instKP8BtnAct.old.kp8Config[9].mode[3] := TRUE;
   instKP8BtnAct.old.kp8Config[9].mode[7] := TRUE;
   instKP8BtnAct.old.kp8Config[10].activate[3] := TRUE;
   instKP8BtnAct.old.kp8Config[10].activate[6] := TRUE;
   instKP8BtnAct.old.kp8Config[10].activate[7] := TRUE;
   instKP8BtnAct.old.kp8Config[10].colorOn1[0] := 'off';
   instKP8BtnAct.old.kp8Config[10].colorOn1[1] := 'off';
   instKP8BtnAct.old.kp8Config[10].colorOn1[2] := 'off';
   instKP8BtnAct.old.kp8Config[10].colorOn1[3] := 'yellow';
   instKP8BtnAct.old.kp8Config[10].colorOn1[4] := 'off';
   instKP8BtnAct.old.kp8Config[10].colorOn1[5] := 'off';
   instKP8BtnAct.old.kp8Config[10].colorOn1[6] := 'yellow';
   instKP8BtnAct.old.kp8Config[10].colorOn1[7] := 'yellow';
   instKP8BtnAct.old.kp8Config[10].colorOn2[0] := 'off';
   instKP8BtnAct.old.kp8Config[10].colorOn2[1] := 'off';
   instKP8BtnAct.old.kp8Config[10].colorOn2[2] := 'off';
   instKP8BtnAct.old.kp8Config[10].colorOn2[4] := 'off';
   instKP8BtnAct.old.kp8Config[10].colorOn2[5] := 'off';
   instKP8BtnAct.old.kp8Config[10].colorOff[0] := 'off';
   instKP8BtnAct.old.kp8Config[10].colorOff[1] := 'off';
   instKP8BtnAct.old.kp8Config[10].colorOff[2] := 'off';
   instKP8BtnAct.old.kp8Config[10].colorOff[3] := 'green';
   instKP8BtnAct.old.kp8Config[10].colorOff[4] := 'off';
   instKP8BtnAct.old.kp8Config[10].colorOff[5] := 'off';
   instKP8BtnAct.old.kp8Config[10].colorOff[6] := 'green';
   instKP8BtnAct.old.kp8Config[10].colorOff[7] := 'green';
   instKP8BtnAct.old.kp8Config[10].mode[3] := TRUE;
   instKP8BtnAct.old.kp8Config[10].mode[6] := TRUE;
   instKP8BtnAct.old.kp8Config[10].mode[7] := TRUE;
   instKP8BtnAct.old.kp8Config[11].activate[3] := TRUE;
   instKP8BtnAct.old.kp8Config[11].activate[6] := TRUE;
   instKP8BtnAct.old.kp8Config[11].activate[7] := TRUE;
   instKP8BtnAct.old.kp8Config[11].colorOn1[0] := 'off';
   instKP8BtnAct.old.kp8Config[11].colorOn1[1] := 'off';
   instKP8BtnAct.old.kp8Config[11].colorOn1[2] := 'off';
   instKP8BtnAct.old.kp8Config[11].colorOn1[3] := 'yellow';
   instKP8BtnAct.old.kp8Config[11].colorOn1[4] := 'off';
   instKP8BtnAct.old.kp8Config[11].colorOn1[5] := 'off';
   instKP8BtnAct.old.kp8Config[11].colorOn1[6] := 'yellow';
   instKP8BtnAct.old.kp8Config[11].colorOn1[7] := 'yellow';
   instKP8BtnAct.old.kp8Config[11].colorOn2[0] := 'off';
   instKP8BtnAct.old.kp8Config[11].colorOn2[1] := 'off';
   instKP8BtnAct.old.kp8Config[11].colorOn2[2] := 'off';
   instKP8BtnAct.old.kp8Config[11].colorOn2[4] := 'off';
   instKP8BtnAct.old.kp8Config[11].colorOn2[5] := 'off';
   instKP8BtnAct.old.kp8Config[11].colorOff[0] := 'off';
   instKP8BtnAct.old.kp8Config[11].colorOff[1] := 'off';
   instKP8BtnAct.old.kp8Config[11].colorOff[2] := 'off';
   instKP8BtnAct.old.kp8Config[11].colorOff[3] := 'green';
   instKP8BtnAct.old.kp8Config[11].colorOff[4] := 'off';
   instKP8BtnAct.old.kp8Config[11].colorOff[5] := 'off';
   instKP8BtnAct.old.kp8Config[11].colorOff[6] := 'green';
   instKP8BtnAct.old.kp8Config[11].colorOff[7] := 'green';
   instKP8BtnAct.old.kp8Config[11].mode[3] := TRUE;
   instKP8BtnAct.old.kp8Config[11].mode[6] := TRUE;
   instKP8BtnAct.old.kp8Config[11].mode[7] := TRUE;
   instKP8BtnAct.old.kp8Config[12].activate[1] := TRUE;
   instKP8BtnAct.old.kp8Config[12].activate[2] := TRUE;
   instKP8BtnAct.old.kp8Config[12].activate[3] := TRUE;
   instKP8BtnAct.old.kp8Config[12].activate[5] := TRUE;
   instKP8BtnAct.old.kp8Config[12].activate[6] := TRUE;
   instKP8BtnAct.old.kp8Config[12].activate[7] := TRUE;
   instKP8BtnAct.old.kp8Config[12].colorOn1[0] := 'off';
   instKP8BtnAct.old.kp8Config[12].colorOn1[1] := 'yellow';
   instKP8BtnAct.old.kp8Config[12].colorOn1[2] := 'yellow';
   instKP8BtnAct.old.kp8Config[12].colorOn1[3] := 'yellow';
   instKP8BtnAct.old.kp8Config[12].colorOn1[4] := 'off';
   instKP8BtnAct.old.kp8Config[12].colorOn1[5] := 'yellow';
   instKP8BtnAct.old.kp8Config[12].colorOn1[6] := 'yellow';
   instKP8BtnAct.old.kp8Config[12].colorOn1[7] := 'yellow';
   instKP8BtnAct.old.kp8Config[12].colorOn2[0] := 'off';
   instKP8BtnAct.old.kp8Config[12].colorOn2[4] := 'off';
   instKP8BtnAct.old.kp8Config[12].colorOff[0] := 'off';
   instKP8BtnAct.old.kp8Config[12].colorOff[1] := 'green';
   instKP8BtnAct.old.kp8Config[12].colorOff[2] := 'green';
   instKP8BtnAct.old.kp8Config[12].colorOff[3] := 'green';
   instKP8BtnAct.old.kp8Config[12].colorOff[4] := 'off';
   instKP8BtnAct.old.kp8Config[12].colorOff[5] := 'green';
   instKP8BtnAct.old.kp8Config[12].colorOff[6] := 'green';
   instKP8BtnAct.old.kp8Config[12].colorOff[7] := 'green';
   instKP8BtnAct.old.kp8Config[12].mode[1] := TRUE;
   instKP8BtnAct.old.kp8Config[12].mode[2] := TRUE;
   instKP8BtnAct.old.kp8Config[12].mode[3] := TRUE;
   instKP8BtnAct.old.kp8Config[12].mode[5] := TRUE;
   instKP8BtnAct.old.kp8Config[12].mode[6] := TRUE;
   instKP8BtnAct.old.kp8Config[12].mode[7] := TRUE;
   instKP8BtnAct.old.kp8Config[13].activate[2] := TRUE;
   instKP8BtnAct.old.kp8Config[13].activate[3] := TRUE;
   instKP8BtnAct.old.kp8Config[13].activate[6] := TRUE;
   instKP8BtnAct.old.kp8Config[13].activate[7] := TRUE;
   instKP8BtnAct.old.kp8Config[13].colorOn1[0] := 'off';
   instKP8BtnAct.old.kp8Config[13].colorOn1[1] := 'off';
   instKP8BtnAct.old.kp8Config[13].colorOn1[2] := 'yellow';
   instKP8BtnAct.old.kp8Config[13].colorOn1[3] := 'yellow';
   instKP8BtnAct.old.kp8Config[13].colorOn1[4] := 'off';
   instKP8BtnAct.old.kp8Config[13].colorOn1[5] := 'off';
   instKP8BtnAct.old.kp8Config[13].colorOn1[6] := 'yellow';
   instKP8BtnAct.old.kp8Config[13].colorOn1[7] := 'yellow';
   instKP8BtnAct.old.kp8Config[13].colorOn2[0] := 'off';
   instKP8BtnAct.old.kp8Config[13].colorOn2[1] := 'off';
   instKP8BtnAct.old.kp8Config[13].colorOn2[4] := 'off';
   instKP8BtnAct.old.kp8Config[13].colorOn2[5] := 'off';
   instKP8BtnAct.old.kp8Config[13].colorOff[0] := 'off';
   instKP8BtnAct.old.kp8Config[13].colorOff[1] := 'off';
   instKP8BtnAct.old.kp8Config[13].colorOff[2] := 'green';
   instKP8BtnAct.old.kp8Config[13].colorOff[3] := 'green';
   instKP8BtnAct.old.kp8Config[13].colorOff[4] := 'off';
   instKP8BtnAct.old.kp8Config[13].colorOff[5] := 'off';
   instKP8BtnAct.old.kp8Config[13].colorOff[6] := 'green';
   instKP8BtnAct.old.kp8Config[13].colorOff[7] := 'green';
   instKP8BtnAct.old.kp8Config[13].mode[2] := TRUE;
   instKP8BtnAct.old.kp8Config[13].mode[3] := TRUE;
   instKP8BtnAct.old.kp8Config[13].mode[6] := TRUE;
   instKP8BtnAct.old.kp8Config[13].mode[7] := TRUE;
   instKP8BtnAct.old.kp8Config[14].activate[2] := TRUE;
   instKP8BtnAct.old.kp8Config[14].activate[3] := TRUE;
   instKP8BtnAct.old.kp8Config[14].activate[5] := TRUE;
   instKP8BtnAct.old.kp8Config[14].activate[6] := TRUE;
   instKP8BtnAct.old.kp8Config[14].activate[7] := TRUE;
   instKP8BtnAct.old.kp8Config[14].colorOn1[0] := 'off';
   instKP8BtnAct.old.kp8Config[14].colorOn1[1] := 'off';
   instKP8BtnAct.old.kp8Config[14].colorOn1[2] := 'yellow';
   instKP8BtnAct.old.kp8Config[14].colorOn1[3] := 'yellow';
   instKP8BtnAct.old.kp8Config[14].colorOn1[4] := 'off';
   instKP8BtnAct.old.kp8Config[14].colorOn1[5] := 'yellow';
   instKP8BtnAct.old.kp8Config[14].colorOn1[6] := 'yellow';
   instKP8BtnAct.old.kp8Config[14].colorOn1[7] := 'yellow';
   instKP8BtnAct.old.kp8Config[14].colorOn2[0] := 'off';
   instKP8BtnAct.old.kp8Config[14].colorOn2[1] := 'off';
   instKP8BtnAct.old.kp8Config[14].colorOn2[4] := 'off';
   instKP8BtnAct.old.kp8Config[14].colorOff[0] := 'off';
   instKP8BtnAct.old.kp8Config[14].colorOff[1] := 'off';
   instKP8BtnAct.old.kp8Config[14].colorOff[2] := 'green';
   instKP8BtnAct.old.kp8Config[14].colorOff[3] := 'green';
   instKP8BtnAct.old.kp8Config[14].colorOff[4] := 'off';
   instKP8BtnAct.old.kp8Config[14].colorOff[5] := 'green';
   instKP8BtnAct.old.kp8Config[14].colorOff[6] := 'green';
   instKP8BtnAct.old.kp8Config[14].colorOff[7] := 'green';
   instKP8BtnAct.old.kp8Config[14].mode[2] := TRUE;
   instKP8BtnAct.old.kp8Config[14].mode[3] := TRUE;
   instKP8BtnAct.old.kp8Config[14].mode[5] := TRUE;
   instKP8BtnAct.old.kp8Config[14].mode[6] := TRUE;
   instKP8BtnAct.old.kp8Config[14].mode[7] := TRUE;
   instKP8BtnAct.old.kp8Config[15].activate[1] := TRUE;
   instKP8BtnAct.old.kp8Config[15].activate[2] := TRUE;
   instKP8BtnAct.old.kp8Config[15].activate[3] := TRUE;
   instKP8BtnAct.old.kp8Config[15].activate[5] := TRUE;
   instKP8BtnAct.old.kp8Config[15].activate[6] := TRUE;
   instKP8BtnAct.old.kp8Config[15].activate[7] := TRUE;
   instKP8BtnAct.old.kp8Config[15].colorOn1[0] := 'off';
   instKP8BtnAct.old.kp8Config[15].colorOn1[1] := 'yellow';
   instKP8BtnAct.old.kp8Config[15].colorOn1[2] := 'yellow';
   instKP8BtnAct.old.kp8Config[15].colorOn1[3] := 'yellow';
   instKP8BtnAct.old.kp8Config[15].colorOn1[4] := 'off';
   instKP8BtnAct.old.kp8Config[15].colorOn1[5] := 'yellow';
   instKP8BtnAct.old.kp8Config[15].colorOn1[6] := 'yellow';
   instKP8BtnAct.old.kp8Config[15].colorOn1[7] := 'yellow';
   instKP8BtnAct.old.kp8Config[15].colorOn2[0] := 'off';
   instKP8BtnAct.old.kp8Config[15].colorOn2[4] := 'off';
   instKP8BtnAct.old.kp8Config[15].colorOff[0] := 'off';
   instKP8BtnAct.old.kp8Config[15].colorOff[1] := 'green';
   instKP8BtnAct.old.kp8Config[15].colorOff[2] := 'green';
   instKP8BtnAct.old.kp8Config[15].colorOff[3] := 'green';
   instKP8BtnAct.old.kp8Config[15].colorOff[4] := 'off';
   instKP8BtnAct.old.kp8Config[15].colorOff[5] := 'green';
   instKP8BtnAct.old.kp8Config[15].colorOff[6] := 'green';
   instKP8BtnAct.old.kp8Config[15].colorOff[7] := 'green';
   instKP8BtnAct.old.kp8Config[15].mode[1] := TRUE;
   instKP8BtnAct.old.kp8Config[15].mode[2] := TRUE;
   instKP8BtnAct.old.kp8Config[15].mode[3] := TRUE;
   instKP8BtnAct.old.kp8Config[15].mode[5] := TRUE;
   instKP8BtnAct.old.kp8Config[15].mode[6] := TRUE;
   instKP8BtnAct.old.kp8Config[15].mode[7] := TRUE;
   instKP8BtnAct.old.kp8Config[16].activate[3] := TRUE;
   instKP8BtnAct.old.kp8Config[16].activate[7] := TRUE;
   instKP8BtnAct.old.kp8Config[16].colorOn1[0] := 'off';
   instKP8BtnAct.old.kp8Config[16].colorOn1[1] := 'off';
   instKP8BtnAct.old.kp8Config[16].colorOn1[2] := 'off';
   instKP8BtnAct.old.kp8Config[16].colorOn1[3] := 'yellow';
   instKP8BtnAct.old.kp8Config[16].colorOn1[4] := 'off';
   instKP8BtnAct.old.kp8Config[16].colorOn1[5] := 'off';
   instKP8BtnAct.old.kp8Config[16].colorOn1[6] := 'off';
   instKP8BtnAct.old.kp8Config[16].colorOn1[7] := 'yellow';
   instKP8BtnAct.old.kp8Config[16].colorOn2[0] := 'off';
   instKP8BtnAct.old.kp8Config[16].colorOn2[1] := 'off';
   instKP8BtnAct.old.kp8Config[16].colorOn2[2] := 'off';
   instKP8BtnAct.old.kp8Config[16].colorOn2[4] := 'off';
   instKP8BtnAct.old.kp8Config[16].colorOn2[5] := 'off';
   instKP8BtnAct.old.kp8Config[16].colorOn2[6] := 'off';
   instKP8BtnAct.old.kp8Config[16].colorOff[0] := 'off';
   instKP8BtnAct.old.kp8Config[16].colorOff[1] := 'off';
   instKP8BtnAct.old.kp8Config[16].colorOff[2] := 'off';
   instKP8BtnAct.old.kp8Config[16].colorOff[3] := 'green';
   instKP8BtnAct.old.kp8Config[16].colorOff[4] := 'off';
   instKP8BtnAct.old.kp8Config[16].colorOff[5] := 'off';
   instKP8BtnAct.old.kp8Config[16].colorOff[6] := 'off';
   instKP8BtnAct.old.kp8Config[16].colorOff[7] := 'green';
   instKP8BtnAct.old.kp8Config[16].mode[3] := TRUE;
   instKP8BtnAct.old.kp8Config[16].mode[7] := TRUE;
   instKP8BtnAct.old.kp8Config[17].activate[2] := TRUE;
   instKP8BtnAct.old.kp8Config[17].activate[3] := TRUE;
   instKP8BtnAct.old.kp8Config[17].activate[6] := TRUE;
   instKP8BtnAct.old.kp8Config[17].activate[7] := TRUE;
   instKP8BtnAct.old.kp8Config[17].colorOn1[0] := 'off';
   instKP8BtnAct.old.kp8Config[17].colorOn1[1] := 'off';
   instKP8BtnAct.old.kp8Config[17].colorOn1[2] := 'yellow';
   instKP8BtnAct.old.kp8Config[17].colorOn1[3] := 'yellow';
   instKP8BtnAct.old.kp8Config[17].colorOn1[4] := 'off';
   instKP8BtnAct.old.kp8Config[17].colorOn1[5] := 'off';
   instKP8BtnAct.old.kp8Config[17].colorOn1[6] := 'yellow';
   instKP8BtnAct.old.kp8Config[17].colorOn1[7] := 'yellow';
   instKP8BtnAct.old.kp8Config[17].colorOn2[0] := 'off';
   instKP8BtnAct.old.kp8Config[17].colorOn2[1] := 'off';
   instKP8BtnAct.old.kp8Config[17].colorOn2[4] := 'off';
   instKP8BtnAct.old.kp8Config[17].colorOn2[5] := 'off';
   instKP8BtnAct.old.kp8Config[17].colorOff[0] := 'off';
   instKP8BtnAct.old.kp8Config[17].colorOff[1] := 'off';
   instKP8BtnAct.old.kp8Config[17].colorOff[2] := 'green';
   instKP8BtnAct.old.kp8Config[17].colorOff[3] := 'green';
   instKP8BtnAct.old.kp8Config[17].colorOff[4] := 'off';
   instKP8BtnAct.old.kp8Config[17].colorOff[5] := 'off';
   instKP8BtnAct.old.kp8Config[17].colorOff[6] := 'green';
   instKP8BtnAct.old.kp8Config[17].colorOff[7] := 'green';
   instKP8BtnAct.old.kp8Config[17].mode[2] := TRUE;
   instKP8BtnAct.old.kp8Config[17].mode[3] := TRUE;
   instKP8BtnAct.old.kp8Config[17].mode[6] := TRUE;
   instKP8BtnAct.old.kp8Config[17].mode[7] := TRUE;
   instKP8BtnAct.old.kp8Config[18].activate[3] := TRUE;
   instKP8BtnAct.old.kp8Config[18].activate[6] := TRUE;
   instKP8BtnAct.old.kp8Config[18].activate[7] := TRUE;
   instKP8BtnAct.old.kp8Config[18].colorOn1[0] := 'off';
   instKP8BtnAct.old.kp8Config[18].colorOn1[1] := 'off';
   instKP8BtnAct.old.kp8Config[18].colorOn1[2] := 'off';
   instKP8BtnAct.old.kp8Config[18].colorOn1[3] := 'yellow';
   instKP8BtnAct.old.kp8Config[18].colorOn1[4] := 'off';
   instKP8BtnAct.old.kp8Config[18].colorOn1[5] := 'off';
   instKP8BtnAct.old.kp8Config[18].colorOn1[6] := 'yellow';
   instKP8BtnAct.old.kp8Config[18].colorOn1[7] := 'yellow';
   instKP8BtnAct.old.kp8Config[18].colorOn2[0] := 'off';
   instKP8BtnAct.old.kp8Config[18].colorOn2[1] := 'off';
   instKP8BtnAct.old.kp8Config[18].colorOn2[2] := 'off';
   instKP8BtnAct.old.kp8Config[18].colorOn2[4] := 'off';
   instKP8BtnAct.old.kp8Config[18].colorOn2[5] := 'off';
   instKP8BtnAct.old.kp8Config[18].colorOff[0] := 'off';
   instKP8BtnAct.old.kp8Config[18].colorOff[1] := 'off';
   instKP8BtnAct.old.kp8Config[18].colorOff[2] := 'off';
   instKP8BtnAct.old.kp8Config[18].colorOff[3] := 'green';
   instKP8BtnAct.old.kp8Config[18].colorOff[4] := 'off';
   instKP8BtnAct.old.kp8Config[18].colorOff[5] := 'off';
   instKP8BtnAct.old.kp8Config[18].colorOff[6] := 'green';
   instKP8BtnAct.old.kp8Config[18].colorOff[7] := 'green';
   instKP8BtnAct.old.kp8Config[18].mode[3] := TRUE;
   instKP8BtnAct.old.kp8Config[18].mode[6] := TRUE;
   instKP8BtnAct.old.kp8Config[18].mode[7] := TRUE;
   instKP8BtnAct.old.kp8Config[19].activate[1] := TRUE;
   instKP8BtnAct.old.kp8Config[19].activate[2] := TRUE;
   instKP8BtnAct.old.kp8Config[19].activate[3] := TRUE;
   instKP8BtnAct.old.kp8Config[19].activate[5] := TRUE;
   instKP8BtnAct.old.kp8Config[19].activate[6] := TRUE;
   instKP8BtnAct.old.kp8Config[19].activate[7] := TRUE;
   instKP8BtnAct.old.kp8Config[19].colorOn1[0] := 'off';
   instKP8BtnAct.old.kp8Config[19].colorOn1[1] := 'yellow';
   instKP8BtnAct.old.kp8Config[19].colorOn1[2] := 'yellow';
   instKP8BtnAct.old.kp8Config[19].colorOn1[3] := 'yellow';
   instKP8BtnAct.old.kp8Config[19].colorOn1[4] := 'off';
   instKP8BtnAct.old.kp8Config[19].colorOn1[5] := 'yellow';
   instKP8BtnAct.old.kp8Config[19].colorOn1[6] := 'yellow';
   instKP8BtnAct.old.kp8Config[19].colorOn1[7] := 'yellow';
   instKP8BtnAct.old.kp8Config[19].colorOn2[0] := 'off';
   instKP8BtnAct.old.kp8Config[19].colorOn2[4] := 'off';
   instKP8BtnAct.old.kp8Config[19].colorOff[0] := 'off';
   instKP8BtnAct.old.kp8Config[19].colorOff[1] := 'green';
   instKP8BtnAct.old.kp8Config[19].colorOff[2] := 'green';
   instKP8BtnAct.old.kp8Config[19].colorOff[3] := 'green';
   instKP8BtnAct.old.kp8Config[19].colorOff[4] := 'off';
   instKP8BtnAct.old.kp8Config[19].colorOff[5] := 'green';
   instKP8BtnAct.old.kp8Config[19].colorOff[6] := 'green';
   instKP8BtnAct.old.kp8Config[19].colorOff[7] := 'green';
   instKP8BtnAct.old.kp8Config[19].mode[1] := TRUE;
   instKP8BtnAct.old.kp8Config[19].mode[2] := TRUE;
   instKP8BtnAct.old.kp8Config[19].mode[3] := TRUE;
   instKP8BtnAct.old.kp8Config[19].mode[5] := TRUE;
   instKP8BtnAct.old.kp8Config[19].mode[6] := TRUE;
   instKP8BtnAct.old.kp8Config[19].mode[7] := TRUE;
   instKP8BtnAct.old.kp8Config[20].colorOn1[0] := 'off';
   instKP8BtnAct.old.kp8Config[20].colorOn1[1] := 'off';
   instKP8BtnAct.old.kp8Config[20].colorOn1[2] := 'off';
   instKP8BtnAct.old.kp8Config[20].colorOn1[3] := 'off';
   instKP8BtnAct.old.kp8Config[20].colorOn1[4] := 'off';
   instKP8BtnAct.old.kp8Config[20].colorOn1[5] := 'off';
   instKP8BtnAct.old.kp8Config[20].colorOn1[6] := 'off';
   instKP8BtnAct.old.kp8Config[20].colorOn1[7] := 'off';
   instKP8BtnAct.old.kp8Config[20].colorOn2[0] := 'off';
   instKP8BtnAct.old.kp8Config[20].colorOn2[1] := 'off';
   instKP8BtnAct.old.kp8Config[20].colorOn2[2] := 'off';
   instKP8BtnAct.old.kp8Config[20].colorOn2[3] := 'off';
   instKP8BtnAct.old.kp8Config[20].colorOn2[4] := 'off';
   instKP8BtnAct.old.kp8Config[20].colorOn2[5] := 'off';
   instKP8BtnAct.old.kp8Config[20].colorOn2[6] := 'off';
   instKP8BtnAct.old.kp8Config[20].colorOn2[7] := 'off';
   instKP8BtnAct.old.kp8Config[20].colorOff[0] := 'off';
   instKP8BtnAct.old.kp8Config[20].colorOff[1] := 'off';
   instKP8BtnAct.old.kp8Config[20].colorOff[2] := 'off';
   instKP8BtnAct.old.kp8Config[20].colorOff[3] := 'off';
   instKP8BtnAct.old.kp8Config[20].colorOff[4] := 'off';
   instKP8BtnAct.old.kp8Config[20].colorOff[5] := 'off';
   instKP8BtnAct.old.kp8Config[20].colorOff[6] := 'off';
   instKP8BtnAct.old.kp8Config[20].colorOff[7] := 'off';
   instKP8BtnAct.old.kp8Config[21].activate[7] := TRUE;
   instKP8BtnAct.old.kp8Config[21].colorOn1[0] := 'off';
   instKP8BtnAct.old.kp8Config[21].colorOn1[1] := 'off';
   instKP8BtnAct.old.kp8Config[21].colorOn1[2] := 'off';
   instKP8BtnAct.old.kp8Config[21].colorOn1[3] := 'off';
   instKP8BtnAct.old.kp8Config[21].colorOn1[4] := 'off';
   instKP8BtnAct.old.kp8Config[21].colorOn1[5] := 'off';
   instKP8BtnAct.old.kp8Config[21].colorOn1[6] := 'off';
   instKP8BtnAct.old.kp8Config[21].colorOn1[7] := 'yellow';
   instKP8BtnAct.old.kp8Config[21].colorOn2[0] := 'off';
   instKP8BtnAct.old.kp8Config[21].colorOn2[1] := 'off';
   instKP8BtnAct.old.kp8Config[21].colorOn2[2] := 'off';
   instKP8BtnAct.old.kp8Config[21].colorOn2[3] := 'off';
   instKP8BtnAct.old.kp8Config[21].colorOn2[4] := 'off';
   instKP8BtnAct.old.kp8Config[21].colorOn2[5] := 'off';
   instKP8BtnAct.old.kp8Config[21].colorOn2[6] := 'off';
   instKP8BtnAct.old.kp8Config[21].colorOff[0] := 'off';
   instKP8BtnAct.old.kp8Config[21].colorOff[1] := 'off';
   instKP8BtnAct.old.kp8Config[21].colorOff[2] := 'off';
   instKP8BtnAct.old.kp8Config[21].colorOff[3] := 'off';
   instKP8BtnAct.old.kp8Config[21].colorOff[4] := 'off';
   instKP8BtnAct.old.kp8Config[21].colorOff[5] := 'off';
   instKP8BtnAct.old.kp8Config[21].colorOff[6] := 'off';
   instKP8BtnAct.old.kp8Config[21].colorOff[7] := 'green';
   instKP8BtnAct.old.kp8Config[21].mode[7] := TRUE;
   instKP8BtnAct.old.kp8Config[22].activate[3] := TRUE;
   instKP8BtnAct.old.kp8Config[22].activate[6] := TRUE;
   instKP8BtnAct.old.kp8Config[22].activate[7] := TRUE;
   instKP8BtnAct.old.kp8Config[22].colorOn1[0] := 'off';
   instKP8BtnAct.old.kp8Config[22].colorOn1[1] := 'off';
   instKP8BtnAct.old.kp8Config[22].colorOn1[2] := 'off';
   instKP8BtnAct.old.kp8Config[22].colorOn1[3] := 'yellow';
   instKP8BtnAct.old.kp8Config[22].colorOn1[4] := 'off';
   instKP8BtnAct.old.kp8Config[22].colorOn1[5] := 'off';
   instKP8BtnAct.old.kp8Config[22].colorOn1[6] := 'yellow';
   instKP8BtnAct.old.kp8Config[22].colorOn1[7] := 'yellow';
   instKP8BtnAct.old.kp8Config[22].colorOn2[0] := 'off';
   instKP8BtnAct.old.kp8Config[22].colorOn2[1] := 'off';
   instKP8BtnAct.old.kp8Config[22].colorOn2[2] := 'off';
   instKP8BtnAct.old.kp8Config[22].colorOn2[4] := 'off';
   instKP8BtnAct.old.kp8Config[22].colorOn2[5] := 'off';
   instKP8BtnAct.old.kp8Config[22].colorOff[0] := 'off';
   instKP8BtnAct.old.kp8Config[22].colorOff[1] := 'off';
   instKP8BtnAct.old.kp8Config[22].colorOff[2] := 'off';
   instKP8BtnAct.old.kp8Config[22].colorOff[3] := 'green';
   instKP8BtnAct.old.kp8Config[22].colorOff[4] := 'off';
   instKP8BtnAct.old.kp8Config[22].colorOff[5] := 'off';
   instKP8BtnAct.old.kp8Config[22].colorOff[6] := 'green';
   instKP8BtnAct.old.kp8Config[22].colorOff[7] := 'green';
   instKP8BtnAct.old.kp8Config[22].mode[3] := TRUE;
   instKP8BtnAct.old.kp8Config[22].mode[6] := TRUE;
   instKP8BtnAct.old.kp8Config[22].mode[7] := TRUE;
   instKP8BtnAct.old.kp8Config[23].activate[7] := TRUE;
   instKP8BtnAct.old.kp8Config[23].colorOn1[0] := 'off';
   instKP8BtnAct.old.kp8Config[23].colorOn1[1] := 'off';
   instKP8BtnAct.old.kp8Config[23].colorOn1[2] := 'off';
   instKP8BtnAct.old.kp8Config[23].colorOn1[3] := 'off';
   instKP8BtnAct.old.kp8Config[23].colorOn1[4] := 'off';
   instKP8BtnAct.old.kp8Config[23].colorOn1[5] := 'off';
   instKP8BtnAct.old.kp8Config[23].colorOn1[6] := 'off';
   instKP8BtnAct.old.kp8Config[23].colorOn1[7] := 'yellow';
   instKP8BtnAct.old.kp8Config[23].colorOn2[0] := 'off';
   instKP8BtnAct.old.kp8Config[23].colorOn2[1] := 'off';
   instKP8BtnAct.old.kp8Config[23].colorOn2[2] := 'off';
   instKP8BtnAct.old.kp8Config[23].colorOn2[3] := 'off';
   instKP8BtnAct.old.kp8Config[23].colorOn2[4] := 'off';
   instKP8BtnAct.old.kp8Config[23].colorOn2[5] := 'off';
   instKP8BtnAct.old.kp8Config[23].colorOn2[6] := 'off';
   instKP8BtnAct.old.kp8Config[23].colorOff[0] := 'off';
   instKP8BtnAct.old.kp8Config[23].colorOff[1] := 'off';
   instKP8BtnAct.old.kp8Config[23].colorOff[2] := 'off';
   instKP8BtnAct.old.kp8Config[23].colorOff[3] := 'off';
   instKP8BtnAct.old.kp8Config[23].colorOff[4] := 'off';
   instKP8BtnAct.old.kp8Config[23].colorOff[5] := 'off';
   instKP8BtnAct.old.kp8Config[23].colorOff[6] := 'off';
   instKP8BtnAct.old.kp8Config[23].colorOff[7] := 'green';
   instKP8BtnAct.old.kp8Config[23].mode[7] := TRUE;
   instKP8BtnAct.old.kp8Config[24].activate[7] := TRUE;
   instKP8BtnAct.old.kp8Config[24].colorOn1[0] := 'off';
   instKP8BtnAct.old.kp8Config[24].colorOn1[1] := 'off';
   instKP8BtnAct.old.kp8Config[24].colorOn1[2] := 'off';
   instKP8BtnAct.old.kp8Config[24].colorOn1[3] := 'off';
   instKP8BtnAct.old.kp8Config[24].colorOn1[4] := 'off';
   instKP8BtnAct.old.kp8Config[24].colorOn1[5] := 'off';
   instKP8BtnAct.old.kp8Config[24].colorOn1[6] := 'off';
   instKP8BtnAct.old.kp8Config[24].colorOn1[7] := 'yellow';
   instKP8BtnAct.old.kp8Config[24].colorOn2[0] := 'off';
   instKP8BtnAct.old.kp8Config[24].colorOn2[1] := 'off';
   instKP8BtnAct.old.kp8Config[24].colorOn2[2] := 'off';
   instKP8BtnAct.old.kp8Config[24].colorOn2[3] := 'off';
   instKP8BtnAct.old.kp8Config[24].colorOn2[4] := 'off';
   instKP8BtnAct.old.kp8Config[24].colorOn2[5] := 'off';
   instKP8BtnAct.old.kp8Config[24].colorOn2[6] := 'off';
   instKP8BtnAct.old.kp8Config[24].colorOff[0] := 'off';
   instKP8BtnAct.old.kp8Config[24].colorOff[1] := 'off';
   instKP8BtnAct.old.kp8Config[24].colorOff[2] := 'off';
   instKP8BtnAct.old.kp8Config[24].colorOff[3] := 'off';
   instKP8BtnAct.old.kp8Config[24].colorOff[4] := 'off';
   instKP8BtnAct.old.kp8Config[24].colorOff[5] := 'off';
   instKP8BtnAct.old.kp8Config[24].colorOff[6] := 'off';
   instKP8BtnAct.old.kp8Config[24].colorOff[7] := 'green';
   instKP8BtnAct.old.kp8Config[24].mode[7] := TRUE;
   instKP8BtnAct.old.kp8Config[25].activate[1] := TRUE;
   instKP8BtnAct.old.kp8Config[25].activate[2] := TRUE;
   instKP8BtnAct.old.kp8Config[25].activate[6] := TRUE;
   instKP8BtnAct.old.kp8Config[25].activate[7] := TRUE;
   instKP8BtnAct.old.kp8Config[25].colorOn1[0] := 'off';
   instKP8BtnAct.old.kp8Config[25].colorOn1[1] := 'yellow';
   instKP8BtnAct.old.kp8Config[25].colorOn1[2] := 'yellow';
   instKP8BtnAct.old.kp8Config[25].colorOn1[3] := 'off';
   instKP8BtnAct.old.kp8Config[25].colorOn1[4] := 'off';
   instKP8BtnAct.old.kp8Config[25].colorOn1[5] := 'off';
   instKP8BtnAct.old.kp8Config[25].colorOn1[6] := 'yellow';
   instKP8BtnAct.old.kp8Config[25].colorOn1[7] := 'yellow';
   instKP8BtnAct.old.kp8Config[25].colorOn2[0] := 'off';
   instKP8BtnAct.old.kp8Config[25].colorOn2[3] := 'off';
   instKP8BtnAct.old.kp8Config[25].colorOn2[4] := 'off';
   instKP8BtnAct.old.kp8Config[25].colorOn2[5] := 'off';
   instKP8BtnAct.old.kp8Config[25].colorOff[0] := 'off';
   instKP8BtnAct.old.kp8Config[25].colorOff[1] := 'green';
   instKP8BtnAct.old.kp8Config[25].colorOff[2] := 'green';
   instKP8BtnAct.old.kp8Config[25].colorOff[3] := 'off';
   instKP8BtnAct.old.kp8Config[25].colorOff[4] := 'off';
   instKP8BtnAct.old.kp8Config[25].colorOff[5] := 'off';
   instKP8BtnAct.old.kp8Config[25].colorOff[6] := 'green';
   instKP8BtnAct.old.kp8Config[25].colorOff[7] := 'green';
   instKP8BtnAct.old.kp8Config[25].mode[1] := TRUE;
   instKP8BtnAct.old.kp8Config[25].mode[2] := TRUE;
   instKP8BtnAct.old.kp8Config[25].mode[6] := TRUE;
   instKP8BtnAct.old.kp8Config[25].mode[7] := TRUE;
   instKP8BtnAct.old.kp8Config[26].activate[1] := TRUE;
   instKP8BtnAct.old.kp8Config[26].activate[2] := TRUE;
   instKP8BtnAct.old.kp8Config[26].activate[3] := TRUE;
   instKP8BtnAct.old.kp8Config[26].activate[5] := TRUE;
   instKP8BtnAct.old.kp8Config[26].activate[6] := TRUE;
   instKP8BtnAct.old.kp8Config[26].activate[7] := TRUE;
   instKP8BtnAct.old.kp8Config[26].colorOn1[0] := 'off';
   instKP8BtnAct.old.kp8Config[26].colorOn1[1] := 'yellow';
   instKP8BtnAct.old.kp8Config[26].colorOn1[2] := 'yellow';
   instKP8BtnAct.old.kp8Config[26].colorOn1[3] := 'yellow';
   instKP8BtnAct.old.kp8Config[26].colorOn1[4] := 'off';
   instKP8BtnAct.old.kp8Config[26].colorOn1[5] := 'yellow';
   instKP8BtnAct.old.kp8Config[26].colorOn1[6] := 'yellow';
   instKP8BtnAct.old.kp8Config[26].colorOn1[7] := 'yellow';
   instKP8BtnAct.old.kp8Config[26].colorOn2[0] := 'off';
   instKP8BtnAct.old.kp8Config[26].colorOn2[4] := 'off';
   instKP8BtnAct.old.kp8Config[26].colorOff[0] := 'off';
   instKP8BtnAct.old.kp8Config[26].colorOff[1] := 'green';
   instKP8BtnAct.old.kp8Config[26].colorOff[2] := 'green';
   instKP8BtnAct.old.kp8Config[26].colorOff[3] := 'green';
   instKP8BtnAct.old.kp8Config[26].colorOff[4] := 'off';
   instKP8BtnAct.old.kp8Config[26].colorOff[5] := 'green';
   instKP8BtnAct.old.kp8Config[26].colorOff[6] := 'green';
   instKP8BtnAct.old.kp8Config[26].colorOff[7] := 'green';
   instKP8BtnAct.old.kp8Config[26].mode[1] := TRUE;
   instKP8BtnAct.old.kp8Config[26].mode[2] := TRUE;
   instKP8BtnAct.old.kp8Config[26].mode[3] := TRUE;
   instKP8BtnAct.old.kp8Config[26].mode[5] := TRUE;
   instKP8BtnAct.old.kp8Config[26].mode[6] := TRUE;
   instKP8BtnAct.old.kp8Config[26].mode[7] := TRUE;
   instKP8BtnAct.old.kp8Config[27].activate[1] := TRUE;
   instKP8BtnAct.old.kp8Config[27].activate[2] := TRUE;
   instKP8BtnAct.old.kp8Config[27].activate[3] := TRUE;
   instKP8BtnAct.old.kp8Config[27].activate[5] := TRUE;
   instKP8BtnAct.old.kp8Config[27].activate[6] := TRUE;
   instKP8BtnAct.old.kp8Config[27].activate[7] := TRUE;
   instKP8BtnAct.old.kp8Config[27].colorOn1[0] := 'off';
   instKP8BtnAct.old.kp8Config[27].colorOn1[1] := 'yellow';
   instKP8BtnAct.old.kp8Config[27].colorOn1[2] := 'yellow';
   instKP8BtnAct.old.kp8Config[27].colorOn1[3] := 'yellow';
   instKP8BtnAct.old.kp8Config[27].colorOn1[4] := 'off';
   instKP8BtnAct.old.kp8Config[27].colorOn1[5] := 'yellow';
   instKP8BtnAct.old.kp8Config[27].colorOn1[6] := 'yellow';
   instKP8BtnAct.old.kp8Config[27].colorOn1[7] := 'yellow';
   instKP8BtnAct.old.kp8Config[27].colorOn2[0] := 'off';
   instKP8BtnAct.old.kp8Config[27].colorOn2[4] := 'off';
   instKP8BtnAct.old.kp8Config[27].colorOff[0] := 'off';
   instKP8BtnAct.old.kp8Config[27].colorOff[1] := 'green';
   instKP8BtnAct.old.kp8Config[27].colorOff[2] := 'green';
   instKP8BtnAct.old.kp8Config[27].colorOff[3] := 'green';
   instKP8BtnAct.old.kp8Config[27].colorOff[4] := 'off';
   instKP8BtnAct.old.kp8Config[27].colorOff[5] := 'green';
   instKP8BtnAct.old.kp8Config[27].colorOff[6] := 'green';
   instKP8BtnAct.old.kp8Config[27].colorOff[7] := 'green';
   instKP8BtnAct.old.kp8Config[27].mode[1] := TRUE;
   instKP8BtnAct.old.kp8Config[27].mode[2] := TRUE;
   instKP8BtnAct.old.kp8Config[27].mode[3] := TRUE;
   instKP8BtnAct.old.kp8Config[27].mode[5] := TRUE;
   instKP8BtnAct.old.kp8Config[27].mode[6] := TRUE;
   instKP8BtnAct.old.kp8Config[27].mode[7] := TRUE;
   instKP8BtnAct.old.kp8Config[28].activate[1] := TRUE;
   instKP8BtnAct.old.kp8Config[28].activate[3] := TRUE;
   instKP8BtnAct.old.kp8Config[28].activate[6] := TRUE;
   instKP8BtnAct.old.kp8Config[28].activate[7] := TRUE;
   instKP8BtnAct.old.kp8Config[28].colorOn1[0] := 'off';
   instKP8BtnAct.old.kp8Config[28].colorOn1[1] := 'yellow';
   instKP8BtnAct.old.kp8Config[28].colorOn1[2] := 'off';
   instKP8BtnAct.old.kp8Config[28].colorOn1[3] := 'yellow';
   instKP8BtnAct.old.kp8Config[28].colorOn1[4] := 'off';
   instKP8BtnAct.old.kp8Config[28].colorOn1[5] := 'off';
   instKP8BtnAct.old.kp8Config[28].colorOn1[6] := 'yellow';
   instKP8BtnAct.old.kp8Config[28].colorOn1[7] := 'yellow';
   instKP8BtnAct.old.kp8Config[28].colorOn2[0] := 'off';
   instKP8BtnAct.old.kp8Config[28].colorOn2[2] := 'off';
   instKP8BtnAct.old.kp8Config[28].colorOn2[4] := 'off';
   instKP8BtnAct.old.kp8Config[28].colorOn2[5] := 'off';
   instKP8BtnAct.old.kp8Config[28].colorOff[0] := 'off';
   instKP8BtnAct.old.kp8Config[28].colorOff[1] := 'green';
   instKP8BtnAct.old.kp8Config[28].colorOff[2] := 'off';
   instKP8BtnAct.old.kp8Config[28].colorOff[3] := 'green';
   instKP8BtnAct.old.kp8Config[28].colorOff[4] := 'off';
   instKP8BtnAct.old.kp8Config[28].colorOff[5] := 'off';
   instKP8BtnAct.old.kp8Config[28].colorOff[6] := 'green';
   instKP8BtnAct.old.kp8Config[28].colorOff[7] := 'green';
   instKP8BtnAct.old.kp8Config[28].mode[1] := TRUE;
   instKP8BtnAct.old.kp8Config[28].mode[3] := TRUE;
   instKP8BtnAct.old.kp8Config[28].mode[6] := TRUE;
   instKP8BtnAct.old.kp8Config[28].mode[7] := TRUE;
   instKP8BtnAct.old.kp8Config[29].activate[1] := TRUE;
   instKP8BtnAct.old.kp8Config[29].activate[2] := TRUE;
   instKP8BtnAct.old.kp8Config[29].activate[3] := TRUE;
